ABB RAPID module: ProgSide1.mod

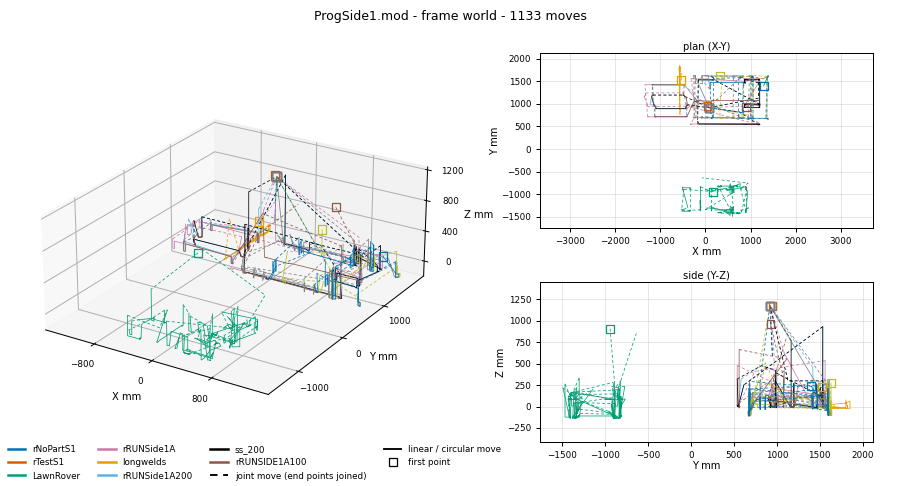
[picture p0: tool path of ProgSide1.mod in frame world, 1133 of 1133 moves have a stored position in this frame; points joined in program order, loops and branches not executed]
MODULE ProgSide1
	PERS bool bZ_B_onlySide2:=FALSE;
	PERS bool bZ_B_onlySide1:=FALSE;
	PERS bool bC_HalfstepSide2:=FALSE;
	PERS bool bC_HalfstepSide1:=FALSE;
	PERS bool bZ_HalfstepSide1:=FALSE;
	PERS bool bZ_HalfstepSide2:=FALSE;
	PERS bool bAngleSide1:=FALSE;
	PERS bool bAngleSide2:=FALSE;
	PERS bool bTestWeldSide1:=FALSE;
    PERS bool bTestWeldSide2:=FALSE;

    ! Boolian initialization for the SS 300 Frames
    PERS bool bNoPartSide1:=FALSE;
	PERS bool bNoPartSide2:=FALSE;
    PERS bool bPart1:=FALSE;
    PERS bool bPart2:=FALSE;
    PERS bool bPart3:=FALSE;
    PERS bool bPart4:=FALSE;
    PERS bool bPart5:=FALSE;
    PERS bool bPart6:=FALSE;
    PERS bool bPart7:=FALSE;
    PERS bool bPart8:=FALSE;
    PERS bool bPart9:=FALSE;
    PERS bool bPart10:=FALSE;
    PERS bool A_onlySide2:=FALSE;
    PERS bool B_onlySide2:=FALSE;
	PERS bool A_onlySide1:=TRUE;
    PERS bool B_onlySide1:=FALSE;
	PERS bool AB_Side1:=FALSE;
    PERS bool AB_Side2:=FALSE;

    ! Boolian initialization for the SelFrames procedures except the SS 300s.
    PERS bool bSkid50:=FALSE;
    PERS bool bSkid100:=FALSE;
	PERS bool bSkid200:=FALSE;
    PERS bool bSide1A100:=FALSE;
    PERS bool bSide1A200:=FALSE;

    PERS bool bRover:=TRUE;
    PERS bool bLongWeld:=FALSE;

    ! Boolian initialization for Parts menu selection.
    PERS bool bPart1:=FALSE;
    PERS bool bPart2:=FALSE;
    PERS bool bPart3:=FALSE;
    PERS bool bPart4:=FALSE;
    PERS bool bPart5:=FALSE;
    PERS bool bPart6:=FALSE;
    PERS bool bPart7:=FALSE;
    PERS bool bPart8:=FALSE;
    PERS bool bPart9:=FALSE;
    PERS bool bPart10:=FALSE;


	TASK PERS welddata weld7:=[15.24,16.6963,[7,0,0,0,0,0,0,0,0],[7,0,0,0,0,0,0,0,0]];
	TASK PERS welddata weld6:=[16.2983,16.6963,[6,0,0,0,0,0,0,0,0],[6,0,0,0,0,0,0,0,0]];

	CONST robtarget pPounceOS1:=[[-398.58,690.45,580.22],[0.00101632,0.999968,-0.00455572,0.00645523],[-1,0,-1,0],[9E+09,9E+09,9E+09,9E+09,9E+09,9E+09]];
	CONST robtarget pPounceS21:=[[580.19,77.23,83.43],[0.071601,0.767336,-0.436334,0.464416],[-1,0,-2,0],[9E+09,9E+09,9E+09,9E+09,9E+09,9E+09]];
	TASK PERS seamdata seam2:=[4,1,[1,0,52,74.0833,0,0,0,0,0],0,0,0,0,0,[1,0,48,0,0,0,0,0,0],0.01,0.1,[1,0,48,105.833,0,0,0,0,0],0,0,[0,0,0,0,0,0,0,0,0],1];
	TASK PERS seamdata seam10:=[4,1,[1,0,50,80.4333,0,0,0,0,0],0,0,0,0,0,[0,0,0,0,0,0,0,0,0],0.25,0.25,[1,0,50,38.1,0,0,0,0,0],0,0,[0,0,0,0,0,0,0,0,0],1];
	CONST robtarget pPounceS31:=[[358.52,159.10,437.93],[0.0181628,-0.398765,0.916866,0.00362624],[-2,0,-2,0],[9E+09,9E+09,9E+09,9E+09,9E+09,9E+09]];
	CONST robtarget pPounceS41:=[[193.25,136.11,113.74],[0.188325,0.84715,-0.195157,0.45693],[-1,-1,-2,0],[9E+09,9E+09,9E+09,9E+09,9E+09,9E+09]];
	PERS welddata weld11:=[13.5467,0,[1,0,50,84.6667,0,0,0,0,0],[0,0,0,0,0,0,0,0,0]];
	PERS welddata weld10:=[14.8167,0,[1,0,50,95.25,0,0,0,0,0],[0,0,0,0,0,0,0,0,0]];
	TASK PERS seamdata seam11:=[1,1,[1,0,50,84.6667,0,0,0,0,0],0,0,0,0,0,[0,0,0,0,0,0,0,0,0],0,0,[0,0,0,0,0,0,0,0,0],0,0,[0,0,0,0,0,0,0,0,0],0];
	TASK PERS seamdata seam12:=[1,1,[1,0,18.5,381,0,0,0,0,0],0,0,0,0,0,[0,0,0,0,0,0,0,0,0],0,0,[0,0,0,0,0,0,0,0,0],0,0,[0,0,0,0,0,0,0,0,0],0];
	TASK PERS seamdata seam13:=[1,1,[1,0,14,127,0,0,0,0,0],0,0,0,0,0,[0,0,0,0,0,0,0,0,0],0,0,[0,0,0,0,0,0,0,0,0],0,0,[0,0,0,0,0,0,0,0,0],0];
	PERS welddata weld12:=[13.97,0,[1,0,50,84.6667,0,0,0,0,0],[0,0,0,0,0,0,0,0,0]];
	PERS welddata weld13:=[6.90033,0,[1,0,20,105.833,0,0,0,0,0],[0,0,0,0,0,0,0,0,0]];
	CONST robtarget pSafeS11:=[[-996.19,963.00,488.78],[0.0459907,-0.688393,0.722625,0.0425673],[1,-1,1,0],[9E+09,9E+09,9E+09,9E+09,9E+09,9E+09]];
	CONST robtarget pSafeS21:=[[-996.19,963.00,488.76],[0.0459983,-0.688397,0.722622,0.0425559],[1,-1,1,0],[9E+09,9E+09,9E+09,9E+09,9E+09,9E+09]];
	CONST robtarget pSafeS31:=[[506.44,675.04,711.34],[0.0314656,-0.935633,0.203865,-0.286426],[0,0,-2,0],[9E+09,9E+09,9E+09,9E+09,9E+09,9E+09]];
	CONST robtarget pSafeS41:=[[488.47,1091.24,654.25],[0.0459806,-0.688392,0.722627,0.0425664],[0,0,-1,0],[9E+09,9E+09,9E+09,9E+09,9E+09,9E+09]];
	CONST robtarget pSafeS51:=[[528.23,1196.89,528.24],[0.224235,-0.753625,-0.525201,-0.325471],[0,-1,-3,0],[9E+09,9E+09,9E+09,9E+09,9E+09,9E+09]];
	CONST robtarget pSafeS61:=[[597.29,1295.03,43.37],[0.191334,-0.732058,-0.538062,-0.371444],[0,-1,-2,0],[9E+09,9E+09,9E+09,9E+09,9E+09,9E+09]];
	CONST robtarget pSafeS71:=[[542.66,1322.39,535.75],[0.223485,-0.764556,-0.487458,-0.357621],[0,-1,-2,0],[9E+09,9E+09,9E+09,9E+09,9E+09,9E+09]];
	CONST robtarget pSafeS81:=[[542.66,1322.38,535.76],[0.223484,-0.764558,-0.487457,-0.35762],[0,-1,-2,0],[9E+09,9E+09,9E+09,9E+09,9E+09,9E+09]];
	CONST robtarget pPounceS51:=[[15.28,993.81,754.75],[0.277209,0.263034,-0.848831,-0.365313],[0,0,0,0],[9E+09,9E+09,9E+09,9E+09,9E+09,9E+09]];
	CONST robtarget pPounceS61:=[[649.55,1131.56,389.19],[0.45355,-0.00505177,-0.879595,-0.143459],[0,0,0,0],[9E+09,9E+09,9E+09,9E+09,9E+09,9E+09]];
	TASK PERS seamdata seam3:=[1,1,[1,0,35,84.6667,0,0,0,0,0],0,0,0,0,0,[1,0,48,0,0,0,0,0,0],0.01,0.1,[1,0,48,105.833,0,0,0,0,0],0,0,[0,0,0,0,0,0,0,0,0],1];
	CONST robtarget pSafeS101:=[[572.94,23.46,738.68],[0.0502756,-0.467207,-0.815726,-0.337314],[0,0,0,0],[9E+09,9E+09,9E+09,9E+09,9E+09,9E+09]];
	CONST robtarget pSafeS111:=[[877.74,-1.14,1156.39],[0.00629855,0.0017594,0.999979,-0.000494623],[0,-1,0,0],[9E+09,9E+09,9E+09,9E+09,9E+09,9E+09]];
	CONST robtarget pSafeS121:=[[877.74,-1.14,1156.39],[0.00629925,0.00175887,0.999979,-0.000492925],[0,-1,0,0],[9E+09,9E+09,9E+09,9E+09,9E+09,9E+09]];
	CONST robtarget pSafeS131:=[[865.02,1139.54,-19.77],[0.144708,-0.274627,0.931028,0.191903],[0,-2,2,0],[9E+09,9E+09,9E+09,9E+09,9E+09,9E+09]];
	CONST robtarget pSafeS141:=[[849.60,1148.97,-24.06],[0.00628216,0.00187497,0.999979,-0.000396021],[0,-1,1,0],[9E+09,9E+09,9E+09,9E+09,9E+09,9E+09]];
	CONST robtarget pSafeS151:=[[1007.97,1505.52,122.27],[0.0460025,-0.688387,0.722632,0.0425454],[0,1,-2,0],[9E+09,9E+09,9E+09,9E+09,9E+09,9E+09]];
	CONST robtarget pHomePos20:=[[365.14,988.92,-33.91],[0.0351389,-0.509982,-0.859022,-0.0276858],[0,-1,1,0],[9E+09,9E+09,9E+09,9E+09,9E+09,9E+09]];
	CONST robtarget pHomePos30:=[[365.15,979.87,-33.91],[0.0351433,-0.509968,-0.85903,-0.0276827],[0,-1,1,0],[9E+09,9E+09,9E+09,9E+09,9E+09,9E+09]];
	CONST robtarget pHomePos40:=[[365.14,979.87,-15.16],[0.0351385,-0.509986,-0.859019,-0.0276867],[0,-1,1,0],[9E+09,9E+09,9E+09,9E+09,9E+09,9E+09]];
	CONST robtarget pHomePos50:=[[433.12,979.73,-15.17],[0.0351369,-0.509964,-0.859032,-0.0276871],[0,-1,1,0],[9E+09,9E+09,9E+09,9E+09,9E+09,9E+09]];
	CONST robtarget pHomePos60:=[[430.57,978.47,-32.25],[0.0351433,-0.50998,-0.859023,-0.0276796],[0,-1,1,0],[9E+09,9E+09,9E+09,9E+09,9E+09,9E+09]];
	CONST robtarget pHomePos70:=[[430.57,978.46,-32.26],[0.0351393,-0.509989,-0.859017,-0.027681],[0,-1,1,0],[9E+09,9E+09,9E+09,9E+09,9E+09,9E+09]];
	CONST robtarget pHomePos80:=[[430.59,974.37,-32.26],[0.0351321,-0.50997,-0.859029,-0.0276862],[0,-1,1,0],[9E+09,9E+09,9E+09,9E+09,9E+09,9E+09]];
	CONST robtarget pHomePos90:=[[430.57,974.36,-24.94],[0.0351397,-0.509992,-0.859016,-0.0276799],[0,-1,1,0],[9E+09,9E+09,9E+09,9E+09,9E+09,9E+09]];
	CONST robtarget pHomePos100:=[[445.83,974.38,-24.94],[0.0351383,-0.509986,-0.859019,-0.0276863],[0,-1,1,0],[9E+09,9E+09,9E+09,9E+09,9E+09,9E+09]];
	CONST robtarget pHomePos110:=[[446.40,974.36,-32.29],[0.0351532,-0.510006,-0.859007,-0.0276708],[0,-1,1,0],[9E+09,9E+09,9E+09,9E+09,9E+09,9E+09]];
	CONST robtarget pHomePos120:=[[446.42,974.37,-32.29],[0.0351424,-0.509994,-0.859014,-0.0276814],[0,-1,1,0],[9E+09,9E+09,9E+09,9E+09,9E+09,9E+09]];
	CONST robtarget pSafeS12:=[[1424.79,-683.57,-13.74],[0.019551,0.168491,0.985501,-0.00412114],[-1,1,-2,0],[9E+09,9E+09,9E+09,9E+09,9E+09,9E+09]];
	CONST robtarget pSafeS22:=[[1462.93,-789.47,-110.40],[0.0637154,0.393325,0.863983,0.307846],[-1,1,-2,0],[9E+09,9E+09,9E+09,9E+09,9E+09,9E+09]];
	CONST robtarget pSafeS32:=[[1462.93,-821.54,-110.39],[0.0637158,0.39332,0.863986,0.307843],[-1,1,-2,0],[9E+09,9E+09,9E+09,9E+09,9E+09,9E+09]];
	CONST robtarget pSafeS42:=[[1462.93,-821.54,-110.39],[0.0637186,0.393326,0.863982,0.307849],[-1,1,-2,0],[9E+09,9E+09,9E+09,9E+09,9E+09,9E+09]];
	CONST robtarget pSafeS52:=[[1462.55,-1477.98,-107.56],[0.0637139,0.393324,0.863983,0.30785],[-1,0,-1,0],[9E+09,9E+09,9E+09,9E+09,9E+09,9E+09]];
	CONST robtarget pSafeS62:=[[1462.54,-1515.56,-107.57],[0.0637098,0.393325,0.863984,0.307846],[-1,0,-1,0],[9E+09,9E+09,9E+09,9E+09,9E+09,9E+09]];
	CONST robtarget pSafeS72:=[[1462.54,-1515.57,-107.57],[0.0637139,0.39333,0.86398,0.307849],[-1,0,-1,0],[9E+09,9E+09,9E+09,9E+09,9E+09,9E+09]];
	CONST robtarget pSafeS82:=[[1462.55,-1515.57,-6.77],[0.063723,0.393334,0.863975,0.307857],[-1,0,-1,0],[9E+09,9E+09,9E+09,9E+09,9E+09,9E+09]];
	CONST robtarget pSafeS161:=[[44.14,948.66,1172.82],[0.0459836,-0.688397,0.722622,0.0425714],[0,-1,0,0],[9E+09,9E+09,9E+09,9E+09,9E+09,9E+09]];
	CONST robtarget pSafeS171:=[[877.68,-1.12,1156.34],[0.00623811,0.00177345,0.999979,-0.000467886],[0,-1,0,0],[9E+09,9E+09,9E+09,9E+09,9E+09,9E+09]];
	CONST robtarget pSafeS181:=[[1178.99,1129.25,299.25],[0.0635535,0.517233,-0.779104,0.348467],[0,1,-3,1],[9E+09,9E+09,9E+09,9E+09,9E+09,9E+09]];
	CONST robtarget pSafeS191:=[[877.68,-1.12,1156.34],[0.00623811,0.00177268,0.999979,-0.000467882],[0,-1,0,0],[9E+09,9E+09,9E+09,9E+09,9E+09,9E+09]];
	CONST robtarget pSafeS201:=[[631.06,-50.80,790.98],[0.377429,-0.0153459,-0.925903,0.00402947],[-1,-1,-5,0],[9E+09,9E+09,9E+09,9E+09,9E+09,9E+09]];
	CONST robtarget pSafeS211:=[[631.06,-50.80,790.98],[0.377429,-0.0153486,-0.925903,0.00403031],[-1,-1,-5,0],[9E+09,9E+09,9E+09,9E+09,9E+09,9E+09]];


!XXXXXXXXXXXXXXXXXXXXXXXXXXXXXXXXXXXXXXXXXXXXXXXXXXXXXXXXXXXX

!XXXXXXXXXXXXXXXXXXXXXXXXXXXXXXXXXXXXXXXXXXXXXXXXXXXXXXXXXXXX
!xxxxxxxxxxxxxxxxxxxxxxxxxxxxxxxxxxxxxxxxxxxxxxxxxxxxxxxxxxxxxxxx




	PROC rNoPartS1()
		MoveJ pSafeS1, v800, fine, tWeldGun;
		MoveJ pPounceS1, v800, fine, tWeldGun;
		MoveJ pSafeS1, v800, fine, tWeldGun;
	ENDPROC
	PROC rTstA1()
		TPWrite "A S1";
	ENDPROC
	PROC rTstB1()
		TPWrite "B S1";
	ENDPROC
	PROC rTestS1()
		MoveJ [[44.14,948.66,1172.81],[0.0459874,-0.688394,0.722625,0.042569],[0,-1,0,0],[9E+09,9E+09,9E+09,9E+09,9E+09,9E+09]], v1000, z50, tWeldGun;
	ENDPROC
	PROC LawnRover()
		rTestPosTop;
		TPWrite "Side 1 B";
		MoveJ [[173.01,-945.09,908.66],[0.230148,-0.640466,-0.674994,-0.284991],[-1,0,0,0],[9E+09,9E+09,9E+09,9E+09,9E+09,9E+09]], vmax, z50, tWeldGun;
		MoveJ [[-516.56,-891.88,262.76],[0.200577,-0.67934,-0.672798,-0.213563],[-2,0,-1,0],[9E+09,9E+09,9E+09,9E+09,9E+09,9E+09]], vmax, z10, tWeldGun;
		MoveL [[-514.49,-897.92,-127.68],[0.230166,-0.665843,-0.672051,-0.22809],[-2,0,-1,0],[9E+09,9E+09,9E+09,9E+09,9E+09,9E+09]], vmax, z10, tWeldGun;
		ArcLStart [[-513.42,-896.95,-136.62],[0.210767,-0.657306,-0.686363,-0.228983],[-2,0,-1,0],[9E+09,9E+09,9E+09,9E+09,9E+09,9E+09]], v50, seam13, weld13\Weave:=weave1, fine, tWeldGun;
		ArcLEnd [[-481.07,-897.11,-138.20],[0.210746,-0.657346,-0.686325,-0.229001],[-2,0,-1,0],[9E+09,9E+09,9E+09,9E+09,9E+09,9E+09]], v5, seam13, weld13\Weave:=weave1, fine, tWeldGun;
		MoveL [[-479.64,-891.87,-91.90],[0.200495,-0.679391,-0.672743,-0.213649],[-2,0,-1,0],[9E+09,9E+09,9E+09,9E+09,9E+09,9E+09]], vmax, z10, tWeldGun;
		MoveJ [[-526.59,-1340.74,-77.97],[0.272049,0.539222,-0.749573,0.270868],[-2,0,-3,0],[9E+09,9E+09,9E+09,9E+09,9E+09,9E+09]], vmax, z10, tWeldGun;
		MoveL [[-519.95,-1336.21,-124.59],[0.179682,0.6848,-0.680507,0.188877],[-2,-1,-3,0],[9E+09,9E+09,9E+09,9E+09,9E+09,9E+09]], vmax, z10, tWeldGun;
		ArcLStart [[-521.69,-1337.70,-132.47],[0.193399,0.681112,-0.684086,0.175244],[-2,-1,-3,0],[9E+09,9E+09,9E+09,9E+09,9E+09,9E+09]], v50, seam13, weld13\Weave:=weave1, fine, tWeldGun;
		ArcLEnd [[-490.93,-1337.53,-132.49],[0.193282,0.681205,-0.684029,0.175234],[-2,-1,-3,0],[9E+09,9E+09,9E+09,9E+09,9E+09,9E+09]], v5, seam13, weld13\Weave:=weave1, fine, tWeldGun;
		MoveL [[-484.84,-1342.71,46.50],[0.235633,0.655478,-0.679432,0.230648],[-2,-1,-3,0],[9E+09,9E+09,9E+09,9E+09,9E+09,9E+09]], vmax, z10, tWeldGun;
		MoveJ [[-392.56,-1296.67,69.52],[0.264192,0.731229,-0.303703,0.550702],[-2,0,0,0],[9E+09,9E+09,9E+09,9E+09,9E+09,9E+09]], vmax, z20, tWeldGun;
		MoveL [[-512.18,-856.47,-124.70],[0.238884,-0.653044,-0.673688,-0.250226],[-2,0,-1,0],[9E+09,9E+09,9E+09,9E+09,9E+09,9E+09]], vmax, z10, tWeldGun;
		ArcLStart [[-513.54,-858.91,-136.72],[0.215398,-0.662814,-0.680722,-0.225612],[-2,0,-1,0],[9E+09,9E+09,9E+09,9E+09,9E+09,9E+09]], v50, seam13, weld13, fine, tWeldGun;
		!ArcLEnd [[-473.42,-859.48,-137.35],[0.215439,-0.662758,-0.68077,-0.22559],[-2,0,-1,0],[9E+09,9E+09,9E+09,9E+09,9E+09,9E+09]], v5, seam13, weld13\Weave:=weave1, fine, tWeldGun;
		!MoveL [[-470.56,-868.46,-128.98],[0.215449,-0.66272,-0.680808,-0.225579],[-2,0,-1,0],[9E+09,9E+09,9E+09,9E+09,9E+09,9E+09]], vmax, z10, tWeldGun;
		!MoveL [[-436.87,-865.82,-129.01],[0.215414,-0.662677,-0.680771,-0.225849],[-2,0,-1,0],[9E+09,9E+09,9E+09,9E+09,9E+09,9E+09]], vmax, z10, tWeldGun;
		!ArcLStart [[-436.92,-859.84,-136.80],[0.215444,-0.662646,-0.680803,-0.225813],[-2,0,-1,0],[9E+09,9E+09,9E+09,9E+09,9E+09,9E+09]], v50, seam13, weld13\Weave:=weave1, fine, tWeldGun;
		!ArcLEnd [[-395.30,-860.19,-135.58],[0.21546,-0.662716,-0.680804,-0.225593],[-2,0,-1,0],[9E+09,9E+09,9E+09,9E+09,9E+09,9E+09]], v5, seam13, weld13\Weave:=weave1, fine, tWeldGun;
		!MoveL [[-394.28,-872.79,-127.38],[0.215463,-0.66272,-0.6808,-0.225589],[-2,0,-1,0],[9E+09,9E+09,9E+09,9E+09,9E+09,9E+09]], vmax, z10, tWeldGun;
		!MoveL [[-366.90,-866.62,-125.77],[0.215457,-0.662713,-0.680808,-0.225591],[-2,0,-1,0],[9E+09,9E+09,9E+09,9E+09,9E+09,9E+09]], vmax, z10, tWeldGun;
		!ArcLStart [[-366.93,-860.65,-137.16],[0.215461,-0.662729,-0.680792,-0.225588],[-2,0,-1,0],[9E+09,9E+09,9E+09,9E+09,9E+09,9E+09]], v50, seam13, weld13\Weave:=weave1, fine, tWeldGun;
		ArcLEnd [[-338.32,-860.21,-136.79],[0.215451,-0.662739,-0.68078,-0.225604],[-2,0,-1,0],[9E+09,9E+09,9E+09,9E+09,9E+09,9E+09]], v5, seam13, weld13\Weave:=weave1, fine, tWeldGun;
		MoveL [[-339.56,-873.86,-125.98],[0.215452,-0.662777,-0.680806,-0.225413],[-2,0,-1,0],[9E+09,9E+09,9E+09,9E+09,9E+09,9E+09]], vmax, z10, tWeldGun;
		MoveL [[-336.25,-871.19,-128.23],[0.0916487,-0.841258,-0.420907,-0.326687],[-2,0,-1,0],[9E+09,9E+09,9E+09,9E+09,9E+09,9E+09]], vmax, z10, tWeldGun;
		ArcLStart [[-338.59,-862.58,-134.25],[0.091653,-0.841261,-0.420909,-0.326675],[-2,0,-1,0],[9E+09,9E+09,9E+09,9E+09,9E+09,9E+09]], v50, seam13, weld13, fine, tWeldGun;
		ArcLEnd [[-343.89,-887.38,-134.91],[0.00905831,0.920106,0.0370212,0.389812],[-2,0,0,0],[9E+09,9E+09,9E+09,9E+09,9E+09,9E+09]], v5, seam13, weld13, fine, tWeldGun;
		MoveL [[-340.52,-888.78,-94.76],[0.0606807,0.91536,0.0671192,0.392339],[-2,0,0,0],[9E+09,9E+09,9E+09,9E+09,9E+09,9E+09]], v100, z10, tWeldGun;
		!MoveL [[-322.29,-862.50,-115.71],[0.124255,-0.837706,-0.434858,-0.306118],[-2,0,0,0],[9E+09,9E+09,9E+09,9E+09,9E+09,9E+09]], v100, z10, tWeldGun;
		!ArcLStart [[-317.89,-862.07,-130.90],[0.120916,-0.838204,-0.433585,-0.307894],[-2,0,0,0],[9E+09,9E+09,9E+09,9E+09,9E+09,9E+09]], v40, seam13, weld13\Weave:=weave1, fine, tWeldGun;
		!ArcLEnd [[-340.01,-859.38,-134.88],[0.124327,-0.837704,-0.434755,-0.306241],[-2,0,0,0],[9E+09,9E+09,9E+09,9E+09,9E+09,9E+09]], v5, seam13, weld13\Weave:=weave1, fine, tWeldGun;
		MoveL [[-337.89,-880.77,33.09],[0.124309,-0.837706,-0.434822,-0.306146],[-2,0,0,0],[9E+09,9E+09,9E+09,9E+09,9E+09,9E+09]], vmax, z10, tWeldGun;
		MoveJ [[-332.34,-1363.85,48.88],[0.219066,0.836756,-0.390875,0.31475],[-2,-1,1,0],[9E+09,9E+09,9E+09,9E+09,9E+09,9E+09]], vmax, z10, tWeldGun;
		MoveL [[-348.32,-1358.04,-125.11],[0.0288552,0.954843,-0.0190534,0.295092],[-2,-1,1,0],[9E+09,9E+09,9E+09,9E+09,9E+09,9E+09]], vmax, z10, tWeldGun;
		ArcLStart [[-348.85,-1357.02,-134.12],[0.0288204,0.95485,-0.0190118,0.295075],[-2,-1,1,0],[9E+09,9E+09,9E+09,9E+09,9E+09,9E+09]], v50, seam13, weld13\Weave:=weave1, fine, tWeldGun;
		ArcLEnd [[-348.77,-1383.12,-133.63],[0.144948,0.917185,-0.235244,0.287092],[-2,-1,1,0],[9E+09,9E+09,9E+09,9E+09,9E+09,9E+09]], v5, seam13, weld13\Weave:=weave1, fine, tWeldGun;
		MoveL [[-352.02,-1382.79,-125.00],[0.145009,0.917103,-0.235465,0.287142],[-2,-1,1,0],[9E+09,9E+09,9E+09,9E+09,9E+09,9E+09]], vmax, z10, tWeldGun;
		!MoveL [[-328.65,-1384.41,-121.55],[0.145003,0.917127,-0.235391,0.287129],[-2,-1,1,0],[9E+09,9E+09,9E+09,9E+09,9E+09,9E+09]], vmax, z10, tWeldGun;
		!ArcLStart [[-329.96,-1384.26,-128.86],[0.144876,0.917192,-0.23532,0.287045],[-2,-1,1,0],[9E+09,9E+09,9E+09,9E+09,9E+09,9E+09]], v40, seam13, weld13\Weave:=weave1, fine, tWeldGun;
		!ArcLEnd [[-349.04,-1384.95,-130.97],[0.144974,0.917151,-0.235337,0.287113],[-2,-1,1,0],[9E+09,9E+09,9E+09,9E+09,9E+09,9E+09]], v5, seam13, weld13\Weave:=weave1, fine, tWeldGun;
		!MoveL [[-350.83,-1367.95,-122.57],[0.144998,0.917131,-0.235387,0.287125],[-2,-1,1,0],[9E+09,9E+09,9E+09,9E+09,9E+09,9E+09]], vmax, z10, tWeldGun;
		MoveL [[-341.99,-1371.18,-117.57],[0.232266,0.668561,-0.669899,0.224308],[-2,-1,1,0],[9E+09,9E+09,9E+09,9E+09,9E+09,9E+09]], vmax, z10, tWeldGun;
		ArcLStart [[-346.14,-1380.75,-134.00],[0.232258,0.668629,-0.669841,0.22429],[-2,-1,1,0],[9E+09,9E+09,9E+09,9E+09,9E+09,9E+09]], v30, seam13, weld13, fine, tWeldGun;
		!ArcLEnd [[-381.42,-1380.96,-134.98],[0.232253,0.668599,-0.669868,0.2243],[-2,-1,1,0],[9E+09,9E+09,9E+09,9E+09,9E+09,9E+09]], v5, seam13, weld13, fine, tWeldGun;
		!MoveL [[-381.43,-1374.36,-128.77],[0.232262,0.668602,-0.669863,0.224299],[-2,-1,1,0],[9E+09,9E+09,9E+09,9E+09,9E+09,9E+09]], vmax, z10, tWeldGun;
		!MoveL [[-417.42,-1374.56,-128.76],[0.232259,0.668611,-0.669855,0.224298],[-2,-1,1,0],[9E+09,9E+09,9E+09,9E+09,9E+09,9E+09]], vmax, z10, tWeldGun;
		!ArcLStart [[-417.85,-1379.53,-134.58],[0.215828,0.673878,-0.675969,0.205846],[-2,-1,1,0],[9E+09,9E+09,9E+09,9E+09,9E+09,9E+09]], v50, seam13, weld13\Weave:=weave1, fine, tWeldGun;
		!ArcLEnd [[-443.05,-1379.79,-134.59],[0.215834,0.673901,-0.675942,0.205854],[-2,-1,1,0],[9E+09,9E+09,9E+09,9E+09,9E+09,9E+09]], v5, seam13, weld13\Weave:=weave1, fine, tWeldGun;
		!MoveL [[-444.47,-1371.57,-127.54],[0.232274,0.66863,-0.669834,0.224288],[-2,-1,1,0],[9E+09,9E+09,9E+09,9E+09,9E+09,9E+09]], vmax, z10, tWeldGun;
		!MoveL [[-474.23,-1371.36,-127.53],[0.232273,0.668635,-0.66983,0.224288],[-2,-1,1,0],[9E+09,9E+09,9E+09,9E+09,9E+09,9E+09]], vmax, z10, tWeldGun;
		!ArcLStart [[-474.48,-1379.73,-135.16],[0.232264,0.668658,-0.669815,0.224273],[-2,-1,1,0],[9E+09,9E+09,9E+09,9E+09,9E+09,9E+09]], v50, seam13, weld13\Weave:=weave1, fine, tWeldGun;
		ArcLEnd [[-520.49,-1380.63,-135.80],[0.232194,0.668749,-0.669754,0.224259],[-2,-1,1,0],[9E+09,9E+09,9E+09,9E+09,9E+09,9E+09]], v5, seam13, weld13\Weave:=weave1, fine, tWeldGun;
		MoveL [[-521.34,-1368.99,120.05],[0.232497,0.668664,-0.669682,0.22441],[-2,-1,1,0],[9E+09,9E+09,9E+09,9E+09,9E+09,9E+09]], vmax, z10, tWeldGun;
		MoveJ [[-94.49,-1349.72,64.27],[0.311518,0.0288903,-0.949685,-0.0148846],[-2,0,-2,0],[9E+09,9E+09,9E+09,9E+09,9E+09,9E+09]], vmax, z10, tWeldGun;
		MoveJ [[-121.47,-1146.91,200.07],[0.233067,0.684788,-0.672515,-0.156426],[-1,-1,-2,0],[9E+09,9E+09,9E+09,9E+09,9E+09,9E+09]], vmax, z10, tWeldGun;
		MoveL [[-117.16,-1374.82,-109.86],[0.220566,0.688799,-0.675571,-0.143216],[-1,-1,-2,0],[9E+09,9E+09,9E+09,9E+09,9E+09,9E+09]], vmax, z10, tWeldGun;
		ArcLStart [[-117.21,-1374.86,-121.15],[0.220636,0.688785,-0.675564,-0.143209],[-1,-1,-2,0],[9E+09,9E+09,9E+09,9E+09,9E+09,9E+09]], v50, seam13, weld13\Weave:=weave1, fine, tWeldGun;
		ArcLEnd [[-117.25,-1343.15,-121.11],[0.220558,0.688816,-0.67554,-0.143296],[-1,-1,-2,0],[9E+09,9E+09,9E+09,9E+09,9E+09,9E+09]], v5, seam13, weld13\Weave:=weave1, fine, tWeldGun;
		MoveL [[-112.47,-1343.13,-110.12],[0.220583,0.6888,-0.675545,-0.143308],[-1,-1,-2,0],[9E+09,9E+09,9E+09,9E+09,9E+09,9E+09]], vmax, z10, tWeldGun;
		MoveL [[-112.47,-861.36,-110.12],[0.220582,0.688805,-0.67554,-0.143307],[-1,-1,-2,0],[9E+09,9E+09,9E+09,9E+09,9E+09,9E+09]], vmax, z10, tWeldGun;
		ArcLStart [[-114.29,-865.15,-124.72],[0.220598,0.688808,-0.675528,-0.143326],[-1,-1,-2,0],[9E+09,9E+09,9E+09,9E+09,9E+09,9E+09]], v50, seam13, weld13\Weave:=weave1, fine, tWeldGun;
		ArcLEnd [[-114.32,-834.89,-124.92],[0.220557,0.688836,-0.675507,-0.143359],[-1,-1,-2,0],[9E+09,9E+09,9E+09,9E+09,9E+09,9E+09]], v5, seam13, weld13\Weave:=weave1, fine, tWeldGun;
		MoveL [[-108.44,-837.80,142.79],[0.0521127,0.721407,-0.690258,0.0200149],[-2,-1,-3,0],[9E+09,9E+09,9E+09,9E+09,9E+09,9E+09]], vmax, z10, tWeldGun;
		MoveJ [[5.08,-892.16,87.65],[0.246917,-0.649526,-0.670091,-0.261011],[-2,0,-1,0],[9E+09,9E+09,9E+09,9E+09,9E+09,9E+09]], vmax, z10, tWeldGun;
		MoveL [[5.70,-898.13,-125.58],[0.246931,-0.64953,-0.670081,-0.261012],[-2,0,-1,0],[9E+09,9E+09,9E+09,9E+09,9E+09,9E+09]], vmax, z10, tWeldGun;
		ArcLStart [[5.30,-897.90,-137.78],[0.203047,-0.669211,-0.681329,-0.216148],[-2,0,-1,0],[9E+09,9E+09,9E+09,9E+09,9E+09,9E+09]], v50, seam13, weld13\Weave:=weave1, fine, tWeldGun;
		ArcLEnd [[39.29,-898.07,-137.00],[0.203054,-0.669216,-0.681319,-0.216158],[-1,0,-1,0],[9E+09,9E+09,9E+09,9E+09,9E+09,9E+09]], v5, seam13, weld13\Weave:=weave1, fine, tWeldGun;
		MoveL [[40.66,-920.62,70.48],[0.246699,-0.649617,-0.670207,-0.260692],[-1,0,-1,0],[9E+09,9E+09,9E+09,9E+09,9E+09,9E+09]], vmax, z10, tWeldGun;
		MoveJ [[283.83,-931.65,13.13],[0.246958,-0.649486,-0.670134,-0.26096],[-1,0,0,0],[9E+09,9E+09,9E+09,9E+09,9E+09,9E+09]], vmax, z10, tWeldGun;
		MoveL [[286.40,-910.85,-115.99],[0.24696,-0.649475,-0.670149,-0.260949],[-1,0,0,0],[9E+09,9E+09,9E+09,9E+09,9E+09,9E+09]], vmax, z10, tWeldGun;
		ArcLStart [[287.09,-901.24,-138.12],[0.20011,-0.665429,-0.68641,-0.214478],[-1,-1,0,0],[9E+09,9E+09,9E+09,9E+09,9E+09,9E+09]], v50, seam13, weld13\Weave:=weave1, fine, tWeldGun;
		ArcLEnd [[319.26,-901.70,-138.51],[0.200189,-0.665343,-0.686488,-0.214425],[-1,-1,0,0],[9E+09,9E+09,9E+09,9E+09,9E+09,9E+09]], v5, seam13, weld13\Weave:=weave1, fine, tWeldGun;
		MoveL [[324.35,-903.06,-116.80],[0.246972,-0.649396,-0.670267,-0.260831],[-1,0,0,0],[9E+09,9E+09,9E+09,9E+09,9E+09,9E+09]], vmax, z10, tWeldGun;
		MoveJ [[559.57,-898.83,-116.82],[0.246966,-0.649476,-0.670148,-0.260944],[-1,-1,0,0],[9E+09,9E+09,9E+09,9E+09,9E+09,9E+09]], vmax, z10, tWeldGun;
		MoveL [[566.73,-906.53,-132.43],[0.246936,-0.649457,-0.670181,-0.260932],[-1,-1,0,0],[9E+09,9E+09,9E+09,9E+09,9E+09,9E+09]], vmax, z10, tWeldGun;
		ArcLStart [[564.18,-902.64,-136.45],[0.203779,-0.664669,-0.684636,-0.219006],[-1,-1,0,0],[9E+09,9E+09,9E+09,9E+09,9E+09,9E+09]], v50, seam13, weld13\Weave:=weave1, fine, tWeldGun;
		ArcLEnd [[595.80,-903.83,-135.82],[0.203773,-0.664709,-0.684589,-0.219037],[-1,-1,0,0],[9E+09,9E+09,9E+09,9E+09,9E+09,9E+09]], v5, seam13, weld13\Weave:=weave1, fine, tWeldGun;
		MoveL [[596.75,-960.43,-56.34],[0.246991,-0.649449,-0.670174,-0.260919],[-1,-1,0,0],[9E+09,9E+09,9E+09,9E+09,9E+09,9E+09]], vmax, z10, tWeldGun;
		MoveJ [[601.82,-903.83,-123.32],[0.326164,-0.613251,-0.630337,-0.346722],[-1,0,0,0],[9E+09,9E+09,9E+09,9E+09,9E+09,9E+09]], vmax, z10, tWeldGun;
		MoveL [[598.73,-903.81,-136.04],[0.274721,-0.639021,-0.654339,-0.296685],[-1,0,0,0],[9E+09,9E+09,9E+09,9E+09,9E+09,9E+09]], v100, z10, tWeldGun;
		ArcLStart [[599.82,-898.69,-137.04],[0.274731,-0.639021,-0.654342,-0.296669],[-1,0,0,0],[9E+09,9E+09,9E+09,9E+09,9E+09,9E+09]], v40, seam13, weld13\Weave:=weave1, fine, tWeldGun;
		ArcLEnd [[632.81,-898.75,-137.05],[0.274699,-0.639022,-0.654363,-0.296649],[-1,0,0,0],[9E+09,9E+09,9E+09,9E+09,9E+09,9E+09]], v5, seam13, weld13\Weave:=weave1, fine, tWeldGun;
		MoveL [[633.74,-910.04,-132.93],[0.326202,-0.613258,-0.630325,-0.346695],[-1,0,0,0],[9E+09,9E+09,9E+09,9E+09,9E+09,9E+09]], vmax, z10, tWeldGun;
		MoveL [[633.73,-910.04,183.03],[0.326216,-0.613247,-0.630334,-0.346685],[-1,0,0,0],[9E+09,9E+09,9E+09,9E+09,9E+09,9E+09]], vmax, z10, tWeldGun;
		MoveJ [[627.00,-822.44,298.30],[0.361159,0.600904,-0.609737,0.36973],[-1,-1,-2,0],[9E+09,9E+09,9E+09,9E+09,9E+09,9E+09]], vmax, z10, tWeldGun;
		MoveL [[627.73,-843.08,-138.79],[0.402411,0.574308,-0.586575,0.405173],[-1,-2,-1,0],[9E+09,9E+09,9E+09,9E+09,9E+09,9E+09]], vmax, z10, tWeldGun;
		ArcLStart [[625.49,-849.82,-138.90],[0.402522,0.574183,-0.586614,0.405185],[-1,-2,-1,0],[9E+09,9E+09,9E+09,9E+09,9E+09,9E+09]], v50, seam13, weld13\Weave:=weave1, fine, tWeldGun;
		ArcLEnd [[591.69,-849.46,-138.90],[0.402522,0.574182,-0.586613,0.405187],[-1,-2,-1,0],[9E+09,9E+09,9E+09,9E+09,9E+09,9E+09]], v5, seam13, weld13\Weave:=weave1, fine, tWeldGun;
		MoveL [[595.98,-827.09,-135.34],[0.402393,0.574513,-0.586267,0.405347],[-1,-2,-1,0],[9E+09,9E+09,9E+09,9E+09,9E+09,9E+09]], vmax, z10, tWeldGun;
		MoveL [[627.09,-846.85,78.98],[0.483059,0.507565,-0.528798,0.478963],[-1,-2,-1,0],[9E+09,9E+09,9E+09,9E+09,9E+09,9E+09]], vmax, z10, tWeldGun;
		ArcLStart [[623.92,-856.82,80.37],[0.483064,0.507539,-0.52884,0.478939],[-1,-2,-1,0],[9E+09,9E+09,9E+09,9E+09,9E+09,9E+09]], v40, seam13, weld13\Weave:=weave1, fine, tWeldGun;
		ArcLEnd [[590.91,-852.32,80.98],[0.483106,0.507553,-0.528792,0.478934],[-1,-2,-1,0],[9E+09,9E+09,9E+09,9E+09,9E+09,9E+09]], v5, seam13, weld13\Weave:=weave1, fine, tWeldGun;
		MoveL [[594.84,-840.41,79.51],[0.487671,0.503288,-0.532967,0.474157],[-1,-2,-1,0],[9E+09,9E+09,9E+09,9E+09,9E+09,9E+09]], vmax, z10, tWeldGun;
		SingArea\Wrist;
		MoveJ [[510.38,-859.01,160.69],[0.00485322,0.746032,-0.024255,0.665452],[-1,0,0,0],[9E+09,9E+09,9E+09,9E+09,9E+09,9E+09]], vmax, z10, tWeldGun;
		MoveL [[590.96,-857.11,78.44],[0.00482135,0.745929,-0.024224,0.665567],[-1,0,0,0],[9E+09,9E+09,9E+09,9E+09,9E+09,9E+09]], vmax, z10, tWeldGun;
		ArcLStart [[595.46,-855.56,78.39],[0.00479068,0.745947,-0.0242061,0.665549],[-1,0,0,0],[9E+09,9E+09,9E+09,9E+09,9E+09,9E+09]], v40, seam13, weld13\Weave:=weave1, fine, tWeldGun;
		ArcLEnd [[594.74,-887.31,78.36],[0.00476122,0.74597,-0.0241871,0.665524],[-1,0,0,0],[9E+09,9E+09,9E+09,9E+09,9E+09,9E+09]], v5, seam13, weld13\Weave:=weave1, fine, tWeldGun;
		MoveL [[545.64,-889.59,83.73],[0.0047987,0.745982,-0.0242261,0.665508],[-1,0,0,0],[9E+09,9E+09,9E+09,9E+09,9E+09,9E+09]], vmax, z10, tWeldGun;
		MoveL [[545.47,-1007.73,83.69],[0.00477345,0.745999,-0.0242032,0.665491],[-1,0,0,0],[9E+09,9E+09,9E+09,9E+09,9E+09,9E+09]], vmax, z10, tWeldGun;
		MoveJ [[631.13,-962.99,83.64],[0.467638,-0.538268,-0.512971,-0.477958],[-1,0,0,0],[9E+09,9E+09,9E+09,9E+09,9E+09,9E+09]], vmax, z10, tWeldGun;
		MoveL [[598.78,-893.01,80.08],[0.467241,-0.531733,-0.519718,-0.478373],[-1,0,0,0],[9E+09,9E+09,9E+09,9E+09,9E+09,9E+09]], vmax, z10, tWeldGun;
		ArcLStart [[597.51,-884.44,80.09],[0.467289,-0.531729,-0.519697,-0.478352],[-1,0,0,0],[9E+09,9E+09,9E+09,9E+09,9E+09,9E+09]], v50, seam13, weld13\Weave:=weave1, fine, tWeldGun;
		ArcLEnd [[628.34,-885.62,79.45],[0.467277,-0.53174,-0.519666,-0.478386],[-1,0,0,0],[9E+09,9E+09,9E+09,9E+09,9E+09,9E+09]], v5, seam13, weld13\Weave:=weave1, fine, tWeldGun;
		MoveL [[633.84,-953.29,84.81],[0.467086,-0.531839,-0.51974,-0.478381],[-1,0,0,0],[9E+09,9E+09,9E+09,9E+09,9E+09,9E+09]], vmax, z10, tWeldGun;
		MoveJ [[-0.34,-1346.80,171.20],[0.287604,0.644423,-0.651566,0.278325],[-1,-1,-2,0],[9E+09,9E+09,9E+09,9E+09,9E+09,9E+09]], vmax, z10, tWeldGun;
		MoveL [[-2.14,-1338.76,-121.61],[0.287464,0.644565,-0.651541,0.278198],[-1,-1,-2,0],[9E+09,9E+09,9E+09,9E+09,9E+09,9E+09]], vmax, z10, tWeldGun;
		ArcLStart [[-0.59,-1345.37,-136.31],[0.245261,0.661538,-0.666169,0.241731],[-1,0,-2,0],[9E+09,9E+09,9E+09,9E+09,9E+09,9E+09]], v40, seam13, weld13\Weave:=weave1, fine, tWeldGun;
		ArcLEnd [[34.33,-1344.96,-135.32],[0.245262,0.661569,-0.666134,0.241742],[-1,0,-2,0],[9E+09,9E+09,9E+09,9E+09,9E+09,9E+09]], v5, seam13, weld13\Weave:=weave1, fine, tWeldGun;
		MoveL [[33.45,-1306.76,35.10],[0.287609,0.644475,-0.651512,0.278328],[-1,-1,-2,0],[9E+09,9E+09,9E+09,9E+09,9E+09,9E+09]], vmax, z10, tWeldGun;
		MoveL [[273.41,-1327.02,35.12],[0.287608,0.6445,-0.651487,0.278327],[-1,-1,-2,0],[9E+09,9E+09,9E+09,9E+09,9E+09,9E+09]], vmax, z10, tWeldGun;
		MoveL [[281.49,-1342.97,-129.04],[0.226085,0.668734,-0.671173,0.226292],[-1,0,-2,0],[9E+09,9E+09,9E+09,9E+09,9E+09,9E+09]], vmax, z10, tWeldGun;
		ArcLStart [[279.86,-1346.54,-134.30],[0.226103,0.668741,-0.671174,0.226249],[-1,0,-2,0],[9E+09,9E+09,9E+09,9E+09,9E+09,9E+09]], v40, seam13, weld13\Weave:=weave1, fine, tWeldGun;
		ArcLEnd [[313.73,-1346.47,-133.85],[0.216577,0.67052,-0.675561,0.217062],[-1,0,-2,0],[9E+09,9E+09,9E+09,9E+09,9E+09,9E+09]], v5, seam13, weld13\Weave:=weave1, fine, tWeldGun;
		MoveL [[313.56,-1350.36,-117.72],[0.287596,0.644518,-0.651477,0.278324],[-1,-1,-2,0],[9E+09,9E+09,9E+09,9E+09,9E+09,9E+09]], vmax, z10, tWeldGun;
		MoveL [[559.03,-1342.37,-128.81],[0.261338,0.655204,-0.662463,0.2521],[-1,0,-2,0],[9E+09,9E+09,9E+09,9E+09,9E+09,9E+09]], vmax, z10, tWeldGun;
		ArcLStart [[559.48,-1347.56,-134.32],[0.242704,0.66214,-0.669449,0.233462],[-1,0,-2,0],[9E+09,9E+09,9E+09,9E+09,9E+09,9E+09]], v40, seam13, weld13\Weave:=weave1, fine, tWeldGun;
		ArcLEnd [[590.72,-1348.56,-134.75],[0.242689,0.662054,-0.669527,0.233498],[-1,0,-2,0],[9E+09,9E+09,9E+09,9E+09,9E+09,9E+09]], v5, seam13, weld13\Weave:=weave1, fine, tWeldGun;
		MoveL [[591.10,-1294.92,-96.48],[0.287644,0.644544,-0.6514,0.278391],[-1,-1,-2,0],[9E+09,9E+09,9E+09,9E+09,9E+09,9E+09]], vmax, z10, tWeldGun;
		MoveL [[591.39,-1347.13,-134.61],[0.309685,0.644241,-0.632283,0.298777],[-1,-1,-2,0],[9E+09,9E+09,9E+09,9E+09,9E+09,9E+09]], vmax, z10, tWeldGun;
		ArcLStart [[596.97,-1352.85,-136.25],[0.320366,0.639208,-0.626493,0.310301],[-1,-1,-2,0],[9E+09,9E+09,9E+09,9E+09,9E+09,9E+09]], v40, seam13, weld13\Weave:=weave1, fine, tWeldGun;
		ArcLEnd [[621.87,-1354.95,-137.78],[0.327716,0.635456,-0.623102,0.317085],[-1,-1,-2,0],[9E+09,9E+09,9E+09,9E+09,9E+09,9E+09]], v5, seam13, weld13\Weave:=weave1, fine, tWeldGun;
		MoveL [[594.26,-1304.04,-124.90],[0.375061,0.603881,-0.605571,0.35769],[-1,-1,-2,0],[9E+09,9E+09,9E+09,9E+09,9E+09,9E+09]], vmax, z10, tWeldGun;
		MoveL [[623.93,-1279.28,49.33],[0.327728,0.635484,-0.623033,0.31715],[-1,-1,-2,0],[9E+09,9E+09,9E+09,9E+09,9E+09,9E+09]], vmax, z10, tWeldGun;
		MoveJ [[598.90,-1494.47,216.89],[0.17643,-0.701594,-0.668329,-0.173135],[-1,-1,0,0],[9E+09,9E+09,9E+09,9E+09,9E+09,9E+09]], vmax, z10, tWeldGun;
		MoveL [[597.59,-1416.16,-134.75],[0.380292,-0.610593,-0.58263,-0.378282],[-1,0,0,0],[9E+09,9E+09,9E+09,9E+09,9E+09,9E+09]], vmax, z10, tWeldGun;
		ArcLStart [[597.06,-1403.16,-135.36],[0.380481,-0.610502,-0.582596,-0.37829],[-1,0,0,0],[9E+09,9E+09,9E+09,9E+09,9E+09,9E+09]], v50, seam13, weld13\Weave:=weave1, fine, tWeldGun;
		ArcLEnd [[627.18,-1403.07,-135.15],[0.380451,-0.610562,-0.582465,-0.378426],[-1,0,0,0],[9E+09,9E+09,9E+09,9E+09,9E+09,9E+09]], v5, seam13, weld13\Weave:=weave1, fine, tWeldGun;
		MoveL [[628.35,-1412.36,-131.21],[0.467542,-0.524114,-0.539124,-0.464817],[-1,0,0,0],[9E+09,9E+09,9E+09,9E+09,9E+09,9E+09]], vmax, z10, tWeldGun;
		MoveL [[630.04,-1413.39,82.24],[0.406954,-0.557371,-0.567573,-0.448985],[-1,0,0,0],[9E+09,9E+09,9E+09,9E+09,9E+09,9E+09]], vmax, z10, tWeldGun;
		ArcLStart [[626.04,-1395.35,81.99],[0.440579,-0.565277,-0.538288,-0.443394],[-1,0,0,0],[9E+09,9E+09,9E+09,9E+09,9E+09,9E+09]], v40, seam13, weld13\Weave:=weave1, fine, tWeldGun;
		ArcLEnd [[593.22,-1395.33,81.95],[0.440608,-0.565286,-0.538264,-0.443384],[-1,0,0,0],[9E+09,9E+09,9E+09,9E+09,9E+09,9E+09]], v5, seam13, weld13\Weave:=weave1, fine, tWeldGun;
		MoveL [[592.54,-1432.49,82.17],[0.427339,-0.575763,-0.543581,-0.436347],[-1,0,0,0],[9E+09,9E+09,9E+09,9E+09,9E+09,9E+09]], vmax, z10, tWeldGun;
		MoveL [[409.08,-1390.23,81.60],[0.377566,-0.521097,-0.645665,-0.411119],[-1,0,0,0],[9E+09,9E+09,9E+09,9E+09,9E+09,9E+09]], vmax, z10, tWeldGun;
		MoveJ [[483.55,-1400.78,96.25],[0.150969,0.719954,0.110873,0.668268],[-1,0,0,0],[9E+09,9E+09,9E+09,9E+09,9E+09,9E+09]], vmax, z10, tWeldGun;
		MoveL [[586.16,-1400.86,80.98],[0.0313045,0.743014,0.0228137,0.668155],[-1,0,0,0],[9E+09,9E+09,9E+09,9E+09,9E+09,9E+09]], vmax, z10, tWeldGun;
		ArcLStart [[593.68,-1399.47,82.20],[0.0312415,0.743073,0.0227754,0.668093],[-1,0,0,0],[9E+09,9E+09,9E+09,9E+09,9E+09,9E+09]], v50, seam13, weld13\Weave:=weave1, fine, tWeldGun;
		ArcLEnd [[593.72,-1363.60,81.06],[0.0313131,0.743053,0.0226814,0.668115],[-1,0,0,0],[9E+09,9E+09,9E+09,9E+09,9E+09,9E+09]], v5, seam13, weld13\Weave:=weave1, fine, tWeldGun;
		MoveL [[554.18,-1372.28,89.73],[0.15109,0.720146,0.110407,0.668112],[-1,0,0,0],[9E+09,9E+09,9E+09,9E+09,9E+09,9E+09]], vmax, z10, tWeldGun;
		MoveL [[549.71,-1268.25,89.71],[0.151117,0.720151,0.110329,0.668113],[-1,1,0,0],[9E+09,9E+09,9E+09,9E+09,9E+09,9E+09]], vmax, z10, tWeldGun;
		MoveJ [[603.39,-1313.43,143.58],[0.469159,0.533622,-0.523436,0.470269],[-1,-2,3,0],[9E+09,9E+09,9E+09,9E+09,9E+09,9E+09]], vmax, z10, tWeldGun;
		MoveL [[591.28,-1347.97,82.12],[0.473675,0.523571,-0.526883,0.473181],[-1,-2,3,0],[9E+09,9E+09,9E+09,9E+09,9E+09,9E+09]], vmax, z10, tWeldGun;
		ArcLStart [[587.96,-1365.88,81.39],[0.473711,0.523325,-0.527202,0.473062],[-1,-2,3,0],[9E+09,9E+09,9E+09,9E+09,9E+09,9E+09]], v40, seam13, weld13\Weave:=weave1, fine, tWeldGun;
		ArcLEnd [[620.94,-1365.88,81.38],[0.473702,0.523289,-0.527255,0.473052],[-1,-2,3,0],[9E+09,9E+09,9E+09,9E+09,9E+09,9E+09]], v5, seam13, weld13\Weave:=weave1, fine, tWeldGun;
		MoveL [[621.57,-1338.36,83.93],[0.473691,0.523533,-0.526918,0.473168],[-1,-2,3,0],[9E+09,9E+09,9E+09,9E+09,9E+09,9E+09]], vmax, z10, tWeldGun;
		MoveJ [[584.48,-948.55,-60.93],[0.252385,-0.649774,-0.664987,-0.268121],[-1,0,0,0],[9E+09,9E+09,9E+09,9E+09,9E+09,9E+09]], vmax, z10, tWeldGun;
		MoveL [[586.13,-889.04,-107.32],[0.252797,-0.649451,-0.665162,-0.26808],[-1,0,0,0],[9E+09,9E+09,9E+09,9E+09,9E+09,9E+09]], vmax, z10, tWeldGun;
		ArcLStart [[584.57,-887.97,-132.03],[0.253395,-0.649148,-0.665278,-0.267962],[-1,0,0,0],[9E+09,9E+09,9E+09,9E+09,9E+09,9E+09]], v40, seam13, weld13\Weave:=weave1, fine, tWeldGun;
		ArcL [[574.57,-892.86,-134.27],[0.253546,-0.649133,-0.665228,-0.267979],[-1,0,0,0],[9E+09,9E+09,9E+09,9E+09,9E+09,9E+09]], v5, seam13, weld13\Weave:=weave1, z0, tWeldGun;
		ArcL [[475.79,-890.51,-134.53],[0.253539,-0.649165,-0.665195,-0.267991],[-1,0,0,0],[9E+09,9E+09,9E+09,9E+09,9E+09,9E+09]], v5, seam13, weld13\Weave:=weave1, z0, tWeldGun;
		ArcLEnd [[466.55,-879.09,-134.47],[0.253642,-0.649098,-0.665227,-0.267977],[-1,0,0,0],[9E+09,9E+09,9E+09,9E+09,9E+09,9E+09]], v5, seam13, weld13\Weave:=weave1, fine, tWeldGun;
		MoveL [[472.59,-879.09,-111.98],[0.253025,-0.6494,-0.665124,-0.268085],[-1,0,0,0],[9E+09,9E+09,9E+09,9E+09,9E+09,9E+09]], vmax, z10, tWeldGun;
		MoveL [[396.83,-879.33,-105.08],[0.253072,-0.649383,-0.665131,-0.268064],[-1,0,0,0],[9E+09,9E+09,9E+09,9E+09,9E+09,9E+09]], vmax, z10, tWeldGun;
		ArcLStart [[394.25,-876.82,-134.70],[0.258595,-0.647157,-0.667412,-0.262448],[-1,-1,0,0],[9E+09,9E+09,9E+09,9E+09,9E+09,9E+09]], v40, seam13, weld13\Weave:=weave1, fine, tWeldGun;
		ArcL [[381.44,-890.37,-135.06],[0.258791,-0.647168,-0.667273,-0.262579],[-1,-1,0,0],[9E+09,9E+09,9E+09,9E+09,9E+09,9E+09]], v5, seam13, weld13\Weave:=weave1, z0, tWeldGun;
		ArcLEnd [[322.18,-889.35,-135.55],[0.25878,-0.64712,-0.667324,-0.262581],[-1,0,0,0],[9E+09,9E+09,9E+09,9E+09,9E+09,9E+09]], v5, seam13, weld13\Weave:=weave1, fine, tWeldGun;
		MoveL [[322.31,-895.09,-116.44],[0.258649,-0.647181,-0.667323,-0.26256],[-1,0,0,0],[9E+09,9E+09,9E+09,9E+09,9E+09,9E+09]], vmax, z10, tWeldGun;
		MoveL [[273.41,-894.64,-124.57],[0.25314,-0.649501,-0.664982,-0.268082],[-1,0,0,0],[9E+09,9E+09,9E+09,9E+09,9E+09,9E+09]], vmax, z10, tWeldGun;
		ArcLStart [[277.62,-889.74,-135.52],[0.25327,-0.649363,-0.665101,-0.267999],[-1,0,0,0],[9E+09,9E+09,9E+09,9E+09,9E+09,9E+09]], v40, seam13, weld13\Weave:=weave1, fine, tWeldGun;
		ArcLEnd [[220.59,-889.99,-136.94],[0.253257,-0.649434,-0.665002,-0.268085],[-1,0,0,0],[9E+09,9E+09,9E+09,9E+09,9E+09,9E+09]], v5, seam13, weld13\Weave:=weave1, fine, tWeldGun;
		MoveL [[221.58,-928.39,28.18],[0.253244,-0.649506,-0.664879,-0.268227],[-1,0,0,0],[9E+09,9E+09,9E+09,9E+09,9E+09,9E+09]], vmax, z10, tWeldGun;
		MoveL [[149.11,-928.37,24.70],[0.253259,-0.649498,-0.664878,-0.268235],[-1,0,0,0],[9E+09,9E+09,9E+09,9E+09,9E+09,9E+09]], vmax, z10, tWeldGun;
		MoveL [[147.94,-898.55,-125.25],[0.226531,-0.659809,-0.673837,-0.243475],[-1,0,0,0],[9E+09,9E+09,9E+09,9E+09,9E+09,9E+09]], vmax, z10, tWeldGun;
		ArcLStart [[145.94,-889.85,-134.87],[0.226621,-0.659751,-0.673869,-0.243461],[-1,0,0,0],[9E+09,9E+09,9E+09,9E+09,9E+09,9E+09]], v40, seam13, weld13\Weave:=weave1, fine, tWeldGun;
		ArcL [[136.31,-880.56,-133.73],[0.179199,-0.674782,-0.68842,-0.196562],[-1,-1,0,0],[9E+09,9E+09,9E+09,9E+09,9E+09,9E+09]], v5, seam13, weld13\Weave:=weave1, z0, tWeldGun;
		ArcLEnd [[135.53,-866.71,-133.14],[0.179149,-0.674875,-0.688323,-0.196627],[-1,-1,0,0],[9E+09,9E+09,9E+09,9E+09,9E+09,9E+09]], v5, seam13, weld13\Weave:=weave1, fine, tWeldGun;
		MoveL [[135.09,-898.03,-81.67],[0.226532,-0.659739,-0.673982,-0.243263],[-1,0,0,0],[9E+09,9E+09,9E+09,9E+09,9E+09,9E+09]], vmax, z10, tWeldGun;
		MoveJ [[133.84,-1301.69,-30.86],[0.241723,0.664636,-0.669792,0.226294],[-1,-1,-2,0],[9E+09,9E+09,9E+09,9E+09,9E+09,9E+09]], vmax, z10, tWeldGun;
		MoveL [[130.27,-1374.37,-120.54],[0.202113,0.676143,-0.685621,0.178621],[-1,0,-2,0],[9E+09,9E+09,9E+09,9E+09,9E+09,9E+09]], vmax, z10, tWeldGun;
		ArcLStart [[129.21,-1375.14,-130.19],[0.202076,0.676173,-0.685603,0.17862],[-1,0,-2,0],[9E+09,9E+09,9E+09,9E+09,9E+09,9E+09]], v40, seam13, weld13\Weave:=weave1, fine, tWeldGun;
		ArcL [[129.40,-1362.73,-131.77],[0.202045,0.676301,-0.68549,0.178601],[-1,0,-2,0],[9E+09,9E+09,9E+09,9E+09,9E+09,9E+09]], v5, seam13, weld13\Weave:=weave1, z0, tWeldGun;
		ArcLEnd [[141.33,-1351.30,-130.96],[0.202027,0.676304,-0.685497,0.178584],[-1,0,-2,0],[9E+09,9E+09,9E+09,9E+09,9E+09,9E+09]], v5, seam13, weld13\Weave:=weave1, fine, tWeldGun;
		MoveL [[140.84,-1281.82,33.20],[0.241757,0.664658,-0.669788,0.226201],[-1,-1,-2,0],[9E+09,9E+09,9E+09,9E+09,9E+09,9E+09]], vmax, z10, tWeldGun;
		MoveL [[199.15,-1314.71,46.47],[0.241551,0.664904,-0.669698,0.225967],[-1,0,-2,0],[9E+09,9E+09,9E+09,9E+09,9E+09,9E+09]], vmax, z10, tWeldGun;
		MoveL [[212.97,-1340.61,-125.15],[0.241813,0.664699,-0.66974,0.226165],[-1,0,-2,0],[9E+09,9E+09,9E+09,9E+09,9E+09,9E+09]], vmax, z10, tWeldGun;
		ArcLStart [[215.34,-1352.26,-133.17],[0.241825,0.664745,-0.669689,0.226168],[-1,0,-2,0],[9E+09,9E+09,9E+09,9E+09,9E+09,9E+09]], v40, seam13, weld13\Weave:=weave1, fine, tWeldGun;
		ArcLEnd [[270.65,-1353.47,-132.38],[0.241836,0.664718,-0.669712,0.226167],[-1,0,-2,0],[9E+09,9E+09,9E+09,9E+09,9E+09,9E+09]], v5, seam13, weld13\Weave:=weave1, fine, tWeldGun;
		MoveL [[270.66,-1348.41,-112.62],[0.241722,0.664804,-0.669653,0.226213],[-1,0,-2,0],[9E+09,9E+09,9E+09,9E+09,9E+09,9E+09]], vmax, z10, tWeldGun;
		MoveL [[316.82,-1344.16,-112.66],[0.241796,0.664657,-0.669739,0.226309],[-1,0,-2,0],[9E+09,9E+09,9E+09,9E+09,9E+09,9E+09]], vmax, z10, tWeldGun;
		ArcLStart [[315.96,-1353.31,-132.51],[0.241791,0.664741,-0.669685,0.22623],[-1,0,-2,0],[9E+09,9E+09,9E+09,9E+09,9E+09,9E+09]], v40, seam13, weld13\Weave:=weave1, fine, tWeldGun;
		ArcL [[378.49,-1354.48,-133.34],[0.24179,0.664785,-0.669645,0.226217],[-1,0,-2,0],[9E+09,9E+09,9E+09,9E+09,9E+09,9E+09]], v5, seam13, weld13\Weave:=weave1, z0, tWeldGun;
		ArcLEnd [[386.30,-1365.07,-133.55],[0.241806,0.664743,-0.669681,0.226219],[-1,0,-2,0],[9E+09,9E+09,9E+09,9E+09,9E+09,9E+09]], v5, seam13, weld13\Weave:=weave1, fine, tWeldGun;
		MoveL [[388.15,-1371.45,-115.55],[0.241783,0.664794,-0.669629,0.226246],[-1,0,-2,0],[9E+09,9E+09,9E+09,9E+09,9E+09,9E+09]], vmax, z10, tWeldGun;
		MoveL [[460.68,-1363.89,-125.97],[0.241779,0.664811,-0.669612,0.226249],[-1,0,-2,0],[9E+09,9E+09,9E+09,9E+09,9E+09,9E+09]], vmax, z10, tWeldGun;
		ArcLStart [[459.75,-1367.07,-131.60],[0.241795,0.664917,-0.669507,0.226233],[-1,0,-2,0],[9E+09,9E+09,9E+09,9E+09,9E+09,9E+09]], v40, seam13, weld13\Weave:=weave1, fine, tWeldGun;
		ArcL [[471.32,-1354.85,-133.04],[0.241789,0.664914,-0.669523,0.226201],[-1,0,-2,0],[9E+09,9E+09,9E+09,9E+09,9E+09,9E+09]], v5, seam13, weld13\Weave:=weave1, z0, tWeldGun;
		ArcL [[571.50,-1356.03,-133.26],[0.241781,0.664938,-0.669508,0.226183],[-1,0,-2,0],[9E+09,9E+09,9E+09,9E+09,9E+09,9E+09]], v5, seam13, weld13\Weave:=weave1, z0, tWeldGun;
		ArcLEnd [[579.28,-1366.47,-130.48],[0.24184,0.664924,-0.669502,0.226179],[-1,0,-2,0],[9E+09,9E+09,9E+09,9E+09,9E+09,9E+09]], v5, seam13, weld13\Weave:=weave1, fine, tWeldGun;
		MoveL [[580.73,-1359.16,-109.60],[0.211837,0.675037,-0.658293,0.257101],[-1,0,-2,0],[9E+09,9E+09,9E+09,9E+09,9E+09,9E+09]], vmax, z10, tWeldGun;
		MoveL [[580.72,-1333.23,219.73],[0.211837,0.67505,-0.658281,0.257098],[-1,0,-2,0],[9E+09,9E+09,9E+09,9E+09,9E+09,9E+09]], vmax, z10, tWeldGun;
		MoveJ [[285.51,-1411.06,96.42],[0.200981,-0.684372,-0.670688,-0.203517],[-1,-1,0,0],[9E+09,9E+09,9E+09,9E+09,9E+09,9E+09]], vmax, z10, tWeldGun;
		MoveL [[279.17,-1421.93,-119.46],[0.177026,-0.688238,-0.684045,-0.164539],[-1,-1,0,0],[9E+09,9E+09,9E+09,9E+09,9E+09,9E+09]], vmax, z10, tWeldGun;
		ArcLStart [[281.45,-1415.02,-128.28],[0.177385,-0.688168,-0.684016,-0.164566],[-1,-1,0,0],[9E+09,9E+09,9E+09,9E+09,9E+09,9E+09]], v40, seam13, weld13\Weave:=weave1, fine, tWeldGun;
		ArcLEnd [[343.22,-1415.08,-128.29],[0.177414,-0.688148,-0.684031,-0.164558],[-1,-1,0,0],[9E+09,9E+09,9E+09,9E+09,9E+09,9E+09]], v5, seam13, weld13\Weave:=weave1, fine, tWeldGun;
		MoveL [[345.60,-1413.44,-114.91],[0.177186,-0.688241,-0.683983,-0.164611],[-1,-1,0,0],[9E+09,9E+09,9E+09,9E+09,9E+09,9E+09]], vmax, z10, tWeldGun;
		MoveL [[346.28,-1412.31,-127.04],[0.247917,-0.667279,-0.662994,-0.231765],[-1,-1,0,0],[9E+09,9E+09,9E+09,9E+09,9E+09,9E+09]], vmax, z10, tWeldGun;
		ArcLStart [[346.07,-1406.84,-129.30],[0.247993,-0.667283,-0.662971,-0.231741],[-1,-1,0,0],[9E+09,9E+09,9E+09,9E+09,9E+09,9E+09]], v40, seam13, weld13\Weave:=weave1, fine, tWeldGun;
		ArcLEnd [[280.68,-1406.02,-129.12],[0.248008,-0.66729,-0.66296,-0.231735],[-1,-1,0,0],[9E+09,9E+09,9E+09,9E+09,9E+09,9E+09]], v5, seam13, weld13\Weave:=weave1, fine, tWeldGun;
		MoveL [[278.24,-1414.33,-118.08],[0.247841,-0.667243,-0.663091,-0.231675],[-1,-1,0,0],[9E+09,9E+09,9E+09,9E+09,9E+09,9E+09]], vmax, z10, tWeldGun;
		MoveL [[281.30,-1410.99,-125.83],[0.247889,-0.667299,-0.662982,-0.231774],[-1,-1,0,0],[9E+09,9E+09,9E+09,9E+09,9E+09,9E+09]], v200, z10, tWeldGun;
		ArcLStart [[281.21,-1407.29,-131.93],[0.247983,-0.667283,-0.662952,-0.231803],[-1,-1,0,0],[9E+09,9E+09,9E+09,9E+09,9E+09,9E+09]], v40, seam13, weld13\Weave:=weave1, fine, tWeldGun;
		ArcLEnd [[346.15,-1406.93,-131.71],[0.248091,-0.667221,-0.662977,-0.231796],[-1,-1,0,0],[9E+09,9E+09,9E+09,9E+09,9E+09,9E+09]], v5, seam13, weld13\Weave:=weave1, fine, tWeldGun;
		MoveL [[346.31,-1422.77,-122.69],[0.247822,-0.667247,-0.663099,-0.231658],[-1,-1,0,0],[9E+09,9E+09,9E+09,9E+09,9E+09,9E+09]], v200, z10, tWeldGun;
		MoveJ [[748.76,-1435.11,122.90],[0.309636,-0.639534,-0.632199,-0.308944],[-1,0,0,0],[9E+09,9E+09,9E+09,9E+09,9E+09,9E+09]], vmax, z10, tWeldGun;
		MoveL [[713.11,-1431.01,114.74],[0.309534,-0.639554,-0.632247,-0.308909],[-1,0,0,0],[9E+09,9E+09,9E+09,9E+09,9E+09,9E+09]], vmax, z10, tWeldGun;
		ArcLStart [[711.57,-1407.93,114.85],[0.309702,-0.639543,-0.632123,-0.309016],[-1,0,0,0],[9E+09,9E+09,9E+09,9E+09,9E+09,9E+09]], v40, seam13, weld13\Weave:=weave1, fine, tWeldGun;
		ArcLEnd [[692.83,-1407.95,87.57],[0.309767,-0.639507,-0.632187,-0.308892],[-1,0,0,0],[9E+09,9E+09,9E+09,9E+09,9E+09,9E+09]], v5, seam13, weld13\Weave:=weave1, fine, tWeldGun;
		MoveL [[694.62,-1427.85,89.22],[0.309609,-0.639506,-0.63227,-0.308883],[-1,0,0,0],[9E+09,9E+09,9E+09,9E+09,9E+09,9E+09]], v200, z10, tWeldGun;
		MoveL [[713.06,-1431.01,114.71],[0.309564,-0.639548,-0.632251,-0.30888],[-1,0,0,0],[9E+09,9E+09,9E+09,9E+09,9E+09,9E+09]], v200, z10, tWeldGun;
		ArcLStart [[712.95,-1408.22,114.38],[0.309717,-0.639503,-0.632179,-0.308968],[-1,0,0,0],[9E+09,9E+09,9E+09,9E+09,9E+09,9E+09]], v40, seam13, weld13\Weave:=weave1, fine, tWeldGun;
		ArcL [[750.96,-1407.06,114.72],[0.309759,-0.639541,-0.632136,-0.308936],[-1,0,0,0],[9E+09,9E+09,9E+09,9E+09,9E+09,9E+09]], v5, seam13, weld13\Weave:=weave1, z20, tWeldGun;
		ArcL [[757.77,-1407.18,96.42],[0.309876,-0.639582,-0.632001,-0.309009],[-1,0,0,0],[9E+09,9E+09,9E+09,9E+09,9E+09,9E+09]], v5, seam13, weld13\Weave:=weave1, z20, tWeldGun;
		ArcLEnd [[769.81,-1407.71,86.71],[0.309836,-0.639623,-0.63199,-0.308987],[-1,0,0,0],[9E+09,9E+09,9E+09,9E+09,9E+09,9E+09]], v5, seam13, weld13\Weave:=weave1, fine, tWeldGun;
		MoveL [[772.20,-1434.22,91.41],[0.309863,-0.63952,-0.632095,-0.30896],[-1,0,0,0],[9E+09,9E+09,9E+09,9E+09,9E+09,9E+09]], vmax, z10, tWeldGun;
		MoveL [[627.48,-1417.65,-2.71],[0.30978,-0.639664,-0.632044,-0.308849],[-1,0,0,0],[9E+09,9E+09,9E+09,9E+09,9E+09,9E+09]], vmax, z10, tWeldGun;
		ArcLStart [[622.56,-1406.59,-12.22],[0.309929,-0.639535,-0.632206,-0.308635],[-1,0,0,0],[9E+09,9E+09,9E+09,9E+09,9E+09,9E+09]], v40, seam13, weld13\Weave:=weave1, fine, tWeldGun;
		ArcL [[586.80,-1407.81,-64.76],[0.310007,-0.639562,-0.632113,-0.30869],[-1,0,0,0],[9E+09,9E+09,9E+09,9E+09,9E+09,9E+09]], v5, seam13, weld13\Weave:=weave1, z0, tWeldGun;
		ArcLEnd [[547.00,-1408.76,-124.51],[0.310106,-0.639539,-0.632128,-0.308607],[-1,0,0,0],[9E+09,9E+09,9E+09,9E+09,9E+09,9E+09]], v5, seam13, weld13\Weave:=weave1, fine, tWeldGun;
		MoveL [[545.98,-1470.65,-122.68],[0.309529,-0.639772,-0.632153,-0.308653],[-1,0,0,0],[9E+09,9E+09,9E+09,9E+09,9E+09,9E+09]], vmax, z10, tWeldGun;
		MoveL [[546.01,-1470.74,261.49],[0.309463,-0.639811,-0.632171,-0.308601],[-1,0,0,0],[9E+09,9E+09,9E+09,9E+09,9E+09,9E+09]], vmax, z10, tWeldGun;
		MoveJ [[450.72,-1393.79,89.08],[0.00680651,0.918501,-0.0118982,0.395183],[-1,0,-3,0],[9E+09,9E+09,9E+09,9E+09,9E+09,9E+09]], vmax, z10, tWeldGun;
		MoveL [[571.40,-1393.78,20.15],[0.00679519,0.918514,-0.0118615,0.395152],[-1,0,-3,0],[9E+09,9E+09,9E+09,9E+09,9E+09,9E+09]], vmax, z10, tWeldGun;
		ArcLStart [[575.83,-1395.64,7.24],[0.00323578,0.944511,-0.0118289,0.328252],[-1,-1,-3,0],[9E+09,9E+09,9E+09,9E+09,9E+09,9E+09]], v50, seam13, weld13\Weave:=weave1, fine, tWeldGun;
		ArcLEnd [[576.75,-1369.68,7.40],[0.00321436,0.944524,-0.0118118,0.328217],[-1,-1,-3,0],[9E+09,9E+09,9E+09,9E+09,9E+09,9E+09]], v5, seam13, weld13\Weave:=weave1, fine, tWeldGun;
		MoveL [[564.04,-1375.65,36.36],[0.00687019,0.918524,-0.0118557,0.395129],[-1,0,-3,0],[9E+09,9E+09,9E+09,9E+09,9E+09,9E+09]], vmax, z10, tWeldGun;
		MoveJ [[280.70,-816.60,118.66],[0.243228,0.672922,-0.664156,0.216597],[-1,0,-2,0],[9E+09,9E+09,9E+09,9E+09,9E+09,9E+09]], vmax, z10, tWeldGun;
		MoveL [[280.45,-816.02,-119.56],[0.197153,0.688424,-0.669151,0.198599],[-1,0,-2,0],[9E+09,9E+09,9E+09,9E+09,9E+09,9E+09]], vmax, z10, tWeldGun;
		ArcLStart [[280.31,-833.88,-132.23],[0.180282,0.693172,-0.676198,0.172535],[-1,0,-2,0],[9E+09,9E+09,9E+09,9E+09,9E+09,9E+09]], v40, seam13, weld13\Weave:=weave1, fine, tWeldGun;
		ArcLEnd [[342.93,-833.70,-131.64],[0.180266,0.693164,-0.6762,0.172574],[-1,0,-2,0],[9E+09,9E+09,9E+09,9E+09,9E+09,9E+09]], v5, seam13, weld13\Weave:=weave1, fine, tWeldGun;
		MoveL [[342.48,-807.65,-103.06],[0.243058,0.673116,-0.664102,0.216347],[-1,0,-2,0],[9E+09,9E+09,9E+09,9E+09,9E+09,9E+09]], vmax, z10, tWeldGun;
		MoveL [[345.00,-832.65,-129.28],[0.23943,0.676376,-0.664326,0.209427],[-1,0,-2,0],[9E+09,9E+09,9E+09,9E+09,9E+09,9E+09]], vmax, z10, tWeldGun;
		ArcLStart [[344.99,-837.69,-131.04],[0.23944,0.676429,-0.664268,0.209432],[-1,0,-2,0],[9E+09,9E+09,9E+09,9E+09,9E+09,9E+09]], v40, seam13, weld13\Weave:=weave1, fine, tWeldGun;
		ArcLEnd [[279.53,-836.97,-132.08],[0.239403,0.676476,-0.664262,0.20934],[-1,0,-2,0],[9E+09,9E+09,9E+09,9E+09,9E+09,9E+09]], v5, seam13, weld13\Weave:=weave1, fine, tWeldGun;
		MoveL [[282.07,-830.03,-127.27],[0.239368,0.676512,-0.664252,0.209295],[-1,0,-2,0],[9E+09,9E+09,9E+09,9E+09,9E+09,9E+09]], vmax, z10, tWeldGun;
		MoveL [[340.63,-830.01,-127.29],[0.276253,0.663629,-0.647063,0.254147],[-1,-1,-2,0],[9E+09,9E+09,9E+09,9E+09,9E+09,9E+09]], vmax, z10, tWeldGun;
		ArcLStart [[341.79,-839.21,-134.25],[0.276248,0.663637,-0.647056,0.25415],[-1,-1,-2,0],[9E+09,9E+09,9E+09,9E+09,9E+09,9E+09]], v40, seam13, weld13\Weave:=weave1, fine, tWeldGun;
		ArcLEnd [[275.96,-839.30,-134.30],[0.276226,0.663648,-0.647095,0.254046],[-1,-1,-2,0],[9E+09,9E+09,9E+09,9E+09,9E+09,9E+09]], v5, seam13, weld13\Weave:=weave1, fine, tWeldGun;
		MoveL [[278.09,-824.22,-132.32],[0.276187,0.663695,-0.647123,0.253895],[-1,-1,-2,0],[9E+09,9E+09,9E+09,9E+09,9E+09,9E+09]], vmax, z10, tWeldGun;
		MoveL [[714.08,-820.90,116.19],[0.255079,0.669279,-0.660332,0.225751],[-1,0,-2,0],[9E+09,9E+09,9E+09,9E+09,9E+09,9E+09]], vmax, z10, tWeldGun;
		ArcLStart [[711.72,-839.02,114.21],[0.255103,0.669318,-0.660289,0.225732],[-1,0,-2,0],[9E+09,9E+09,9E+09,9E+09,9E+09,9E+09]], v40, seam13, weld13\Weave:=weave1, fine, tWeldGun;
		ArcLEnd [[689.82,-838.03,85.78],[0.255132,0.66942,-0.660194,0.225676],[-1,0,-2,0],[9E+09,9E+09,9E+09,9E+09,9E+09,9E+09]], v5, seam13, weld13\Weave:=weave1, fine, tWeldGun;
		MoveL [[693.54,-821.10,87.96],[0.255102,0.669397,-0.660268,0.225562],[-1,0,-2,0],[9E+09,9E+09,9E+09,9E+09,9E+09,9E+09]], v200, z10, tWeldGun;
		MoveL [[714.11,-820.85,116.18],[0.255054,0.669249,-0.660379,0.225731],[-1,0,-2,0],[9E+09,9E+09,9E+09,9E+09,9E+09,9E+09]], v200, z10, tWeldGun;
		ArcLStart [[712.35,-839.62,114.96],[0.255166,0.669278,-0.660318,0.225695],[-1,0,-2,0],[9E+09,9E+09,9E+09,9E+09,9E+09,9E+09]], v40, seam13, weld13\Weave:=weave1, fine, tWeldGun;
		ArcL [[749.58,-839.57,114.36],[0.255124,0.669325,-0.660279,0.225718],[-1,0,-2,0],[9E+09,9E+09,9E+09,9E+09,9E+09,9E+09]], v5, seam13, weld13\Weave:=weave1, z10, tWeldGun;
		ArcL [[755.54,-839.23,95.73],[0.255123,0.669215,-0.66041,0.225659],[-1,0,-2,0],[9E+09,9E+09,9E+09,9E+09,9E+09,9E+09]], v5, seam13, weld13\Weave:=weave1, z10, tWeldGun;
		ArcLEnd [[767.76,-839.65,85.57],[0.255158,0.669169,-0.660424,0.225719],[-1,0,-2,0],[9E+09,9E+09,9E+09,9E+09,9E+09,9E+09]], v5, seam13, weld13\Weave:=weave1, fine, tWeldGun;
		MoveL [[772.08,-767.27,86.77],[0.255103,0.66918,-0.660433,0.225721],[-1,0,-2,0],[9E+09,9E+09,9E+09,9E+09,9E+09,9E+09]], vmax, z10, tWeldGun;
		MoveL [[627.18,-826.93,-5.83],[0.253508,0.65756,-0.66005,0.26016],[-1,0,-2,0],[9E+09,9E+09,9E+09,9E+09,9E+09,9E+09]], vmax, z10, tWeldGun;
		ArcLStart [[625.59,-838.29,-9.60],[0.253597,0.657512,-0.659967,0.260404],[-1,0,-2,0],[9E+09,9E+09,9E+09,9E+09,9E+09,9E+09]], v40, seam13, weld13\Weave:=weave1, fine, tWeldGun;
		ArcL [[579.59,-838.82,-74.40],[0.253602,0.657534,-0.659951,0.260383],[-1,0,-2,0],[9E+09,9E+09,9E+09,9E+09,9E+09,9E+09]], v5, seam13, weld13\Weave:=weave1, z0, tWeldGun;
		ArcLEnd [[541.11,-838.82,-130.24],[0.253635,0.657488,-0.659927,0.260529],[-1,0,-2,0],[9E+09,9E+09,9E+09,9E+09,9E+09,9E+09]], v5, seam13, weld13\Weave:=weave1, fine, tWeldGun;
		MoveL [[548.88,-773.40,234.33],[0.243177,0.673515,-0.663846,0.215757],[-1,0,-2,0],[9E+09,9E+09,9E+09,9E+09,9E+09,9E+09]], vmax, z10, tWeldGun;
		MoveJ [[554.61,-845.95,234.31],[0.0125503,-0.913958,0.00705174,-0.405554],[-1,0,-3,0],[9E+09,9E+09,9E+09,9E+09,9E+09,9E+09]], vmax, z10, tWeldGun;
		MoveL [[577.03,-856.78,17.59],[0.00389083,-0.924944,0.010701,-0.379933],[-1,-1,-3,0],[9E+09,9E+09,9E+09,9E+09,9E+09,9E+09]], vmax, z10, tWeldGun;
		ArcLStart [[581.29,-855.54,4.69],[0.00394985,-0.924973,0.0105669,-0.379867],[-1,-1,-3,0],[9E+09,9E+09,9E+09,9E+09,9E+09,9E+09]], v40, seam13, weld13\Weave:=weave1, fine, tWeldGun;
		ArcLEnd [[581.36,-879.94,4.55],[0.00400335,-0.924982,0.0105343,-0.379844],[-1,-1,-3,0],[9E+09,9E+09,9E+09,9E+09,9E+09,9E+09]], v5, seam13, weld13\Weave:=weave1, fine, tWeldGun;
		MoveL [[536.09,-886.10,63.12],[0.0125865,-0.913974,0.00698526,-0.405519],[-1,0,-3,0],[9E+09,9E+09,9E+09,9E+09,9E+09,9E+09]], vmax, z10, tWeldGun;
		MoveJ [[471.77,-923.60,234.81],[0.361351,0.15882,-0.917288,0.0527665],[-1,0,-1,0],[9E+09,9E+09,9E+09,9E+09,9E+09,9E+09]], vmax, z10, tWeldGun;
		MoveL [[900.49,-837.79,215.66],[0.339396,0.215461,-0.903746,0.147074],[-1,-1,-1,0],[9E+09,9E+09,9E+09,9E+09,9E+09,9E+09]], vmax, z10, tWeldGun;
		MoveL [[900.44,-837.75,127.43],[0.339421,0.215477,-0.903738,0.147042],[-1,-1,-1,0],[9E+09,9E+09,9E+09,9E+09,9E+09,9E+09]], vmax, z10, tWeldGun;
		ArcLStart [[891.28,-846.19,116.68],[0.339399,0.215507,-0.90374,0.147034],[-1,-1,-1,0],[9E+09,9E+09,9E+09,9E+09,9E+09,9E+09]], v40, seam13, weld13\Weave:=weave1, fine, tWeldGun;
		ArcLEnd [[890.65,-846.37,81.46],[0.339418,0.215511,-0.903735,0.147018],[-1,-1,-1,0],[9E+09,9E+09,9E+09,9E+09,9E+09,9E+09]], v5, seam13, weld13\Weave:=weave1, fine, tWeldGun;
		MoveL [[900.41,-837.71,81.46],[0.339442,0.215511,-0.903726,0.147016],[-1,-1,-1,0],[9E+09,9E+09,9E+09,9E+09,9E+09,9E+09]], vmax, z10, tWeldGun;
		MoveL [[900.39,-837.71,198.80],[0.339465,0.215526,-0.903715,0.147012],[-1,-1,-1,0],[9E+09,9E+09,9E+09,9E+09,9E+09,9E+09]], vmax, z10, tWeldGun;
		MoveJ [[893.27,-898.66,198.53],[0.473399,-0.27429,-0.79444,-0.263675],[-1,0,-1,0],[9E+09,9E+09,9E+09,9E+09,9E+09,9E+09]], vmax, z10, tWeldGun;
		MoveL [[893.26,-898.66,124.83],[0.4734,-0.274289,-0.794437,-0.263683],[-1,0,-1,0],[9E+09,9E+09,9E+09,9E+09,9E+09,9E+09]], vmax, z10, tWeldGun;
		ArcLStart [[887.28,-891.68,117.80],[0.48296,-0.257091,-0.803409,-0.234924],[-1,0,-1,0],[9E+09,9E+09,9E+09,9E+09,9E+09,9E+09]], v40, seam13, weld13\Weave:=weave1, fine, tWeldGun;
		ArcLEnd [[887.29,-891.67,77.79],[0.477055,-0.267897,-0.797911,-0.25296],[-1,0,-1,0],[9E+09,9E+09,9E+09,9E+09,9E+09,9E+09]], v5, seam13, weld13\Weave:=weave1, fine, tWeldGun;
		MoveL [[937.32,-934.77,92.77],[0.477007,-0.267909,-0.797948,-0.252921],[-1,0,-1,0],[9E+09,9E+09,9E+09,9E+09,9E+09,9E+09]], vmax, z10, tWeldGun;
		MoveL [[898.69,-1405.03,162.74],[0.405782,-0.372754,-0.813112,-0.187737],[-1,-1,-1,0],[9E+09,9E+09,9E+09,9E+09,9E+09,9E+09]], vmax, z10, tWeldGun;
		MoveL [[893.71,-1403.99,128.70],[0.405776,-0.37274,-0.81311,-0.187787],[-1,-1,-1,0],[9E+09,9E+09,9E+09,9E+09,9E+09,9E+09]], vmax, z10, tWeldGun;
		ArcLStart [[884.67,-1404.01,118.73],[0.405809,-0.372745,-0.8131,-0.187747],[-1,-1,-1,0],[9E+09,9E+09,9E+09,9E+09,9E+09,9E+09]], v40, seam13, weld13\Weave:=weave1, fine, tWeldGun;
		ArcLEnd [[884.66,-1404.02,87.70],[0.40582,-0.372749,-0.813094,-0.187742],[-1,-1,-1,0],[9E+09,9E+09,9E+09,9E+09,9E+09,9E+09]], v5, seam13, weld13\Weave:=weave1, fine, tWeldGun;
		MoveL [[899.80,-1417.41,147.01],[0.405769,-0.372778,-0.81311,-0.187726],[-1,-1,-1,0],[9E+09,9E+09,9E+09,9E+09,9E+09,9E+09]], vmax, z10, tWeldGun;
		MoveJ [[891.04,-1353.86,172.64],[0.459453,0.258247,-0.822177,0.215029],[-1,-1,-1,0],[9E+09,9E+09,9E+09,9E+09,9E+09,9E+09]], vmax, z10, tWeldGun;
		MoveL [[890.95,-1353.84,123.85],[0.45951,0.258257,-0.822151,0.214995],[-1,-1,-1,0],[9E+09,9E+09,9E+09,9E+09,9E+09,9E+09]], vmax, z10, tWeldGun;
		ArcLStart [[883.98,-1356.19,118.84],[0.459511,0.258226,-0.822164,0.214982],[-1,-1,-1,0],[9E+09,9E+09,9E+09,9E+09,9E+09,9E+09]], v40, seam13, weld13\Weave:=weave1, fine, tWeldGun;
		ArcLEnd [[883.33,-1356.75,82.88],[0.459529,0.258231,-0.822154,0.214972],[-1,-1,-1,0],[9E+09,9E+09,9E+09,9E+09,9E+09,9E+09]], v5, seam13, weld13\Weave:=weave1, fine, tWeldGun;
		MoveL [[954.45,-1305.33,82.88],[0.459526,0.258233,-0.822153,0.21498],[-1,-1,-1,0],[9E+09,9E+09,9E+09,9E+09,9E+09,9E+09]], vmax, z10, tWeldGun;
		MoveL [[954.64,-1305.47,331.71],[0.459382,0.258257,-0.822177,0.215165],[-1,-1,-1,0],[9E+09,9E+09,9E+09,9E+09,9E+09,9E+09]], vmax, z10, tWeldGun;
		MoveJ [[785.08,-1364.00,203.32],[0.00171317,-0.947718,0.00701896,-0.319029],[-1,-1,1,0],[9E+09,9E+09,9E+09,9E+09,9E+09,9E+09]], vmax, z10, tWeldGun;
		MoveL [[803.47,-1368.09,131.07],[0.00412255,-0.937659,0.00608177,-0.347481],[-1,-1,1,0],[9E+09,9E+09,9E+09,9E+09,9E+09,9E+09]], vmax, z10, tWeldGun;
		ArcLStart [[804.13,-1366.42,123.85],[0.00419124,-0.937702,0.00597678,-0.347365],[-1,-1,1,0],[9E+09,9E+09,9E+09,9E+09,9E+09,9E+09]], v40, seam13, weld13\Weave:=weave1, fine, tWeldGun;
		ArcLEnd [[804.13,-1396.73,123.94],[0.00421357,-0.937701,0.00598234,-0.347367],[-1,-1,1,0],[9E+09,9E+09,9E+09,9E+09,9E+09,9E+09]], v5, seam13, weld13\Weave:=weave1, fine, tWeldGun;
		MoveL [[799.72,-1397.77,160.94],[0.00406041,-0.937645,0.00597838,-0.34752],[-1,-1,1,0],[9E+09,9E+09,9E+09,9E+09,9E+09,9E+09]], vmax, z10, tWeldGun;
		MoveJ [[912.45,-910.97,281.24],[0.471963,-0.00834501,-0.88125,-0.0240746],[-1,-1,-1,0],[9E+09,9E+09,9E+09,9E+09,9E+09,9E+09]], vmax, z10, tWeldGun;
		MoveL [[909.26,-887.50,143.89],[0.306131,-0.0105667,-0.951842,-0.0130303],[-1,0,-1,0],[9E+09,9E+09,9E+09,9E+09,9E+09,9E+09]], vmax, z10, tWeldGun;
		ArcLStart [[895.38,-884.91,123.01],[0.306206,-0.0106151,-0.951816,-0.0131321],[-1,0,-1,0],[9E+09,9E+09,9E+09,9E+09,9E+09,9E+09]], v40, seam13, weld13\Weave:=weave1, fine, tWeldGun;
		ArcLEnd [[895.62,-855.31,122.99],[0.306213,-0.0106343,-0.951813,-0.0131465],[-1,0,-1,0],[9E+09,9E+09,9E+09,9E+09,9E+09,9E+09]], v5, seam13, weld13\Weave:=weave1, fine, tWeldGun;
		MoveL [[912.81,-855.15,147.89],[0.30614,-0.0105141,-0.95184,-0.0129908],[-1,0,-1,0],[9E+09,9E+09,9E+09,9E+09,9E+09,9E+09]], vmax, z10, tWeldGun;
		MoveJ [[902.72,-1362.89,137.84],[0.306146,-0.0105253,-0.951838,-0.0129664],[-1,0,-1,0],[9E+09,9E+09,9E+09,9E+09,9E+09,9E+09]], vmax, z10, tWeldGun;
		MoveL [[908.97,-1368.68,133.52],[0.305903,-0.0107467,-0.951921,-0.0124571],[-1,0,-1,0],[9E+09,9E+09,9E+09,9E+09,9E+09,9E+09]], vmax, z10, tWeldGun;
		ArcLStart [[891.85,-1362.07,124.85],[0.305985,-0.010764,-0.951893,-0.0125866],[-1,0,-1,0],[9E+09,9E+09,9E+09,9E+09,9E+09,9E+09]], v40, seam13, weld13\Weave:=weave1, fine, tWeldGun;
		ArcLEnd [[891.60,-1393.64,124.58],[0.306016,-0.0107572,-0.951883,-0.0125206],[-1,0,-1,0],[9E+09,9E+09,9E+09,9E+09,9E+09,9E+09]], v5, seam13, weld13\Weave:=weave1, fine, tWeldGun;
		MoveL [[900.37,-1394.95,165.72],[0.306084,-0.0106333,-0.95186,-0.0127431],[-1,0,-1,0],[9E+09,9E+09,9E+09,9E+09,9E+09,9E+09]], vmax, z10, tWeldGun;
		MoveJ [[778.65,-875.76,193.58],[0.0091964,-0.885136,-0.0131126,-0.465058],[-1,0,1,0],[9E+09,9E+09,9E+09,9E+09,9E+09,9E+09]], vmax, z10, tWeldGun;
		MoveL [[804.53,-888.57,142.41],[0.00795263,-0.941332,-0.0147738,-0.337067],[-1,-1,1,0],[9E+09,9E+09,9E+09,9E+09,9E+09,9E+09]], vmax, z10, tWeldGun;
		ArcLStart [[807.14,-888.84,121.83],[0.0115328,-0.957016,-0.0172521,-0.289293],[-1,-1,1,0],[9E+09,9E+09,9E+09,9E+09,9E+09,9E+09]], v40, seam13, weld13\Weave:=weave1, fine, tWeldGun;
		ArcLEnd [[807.38,-858.36,122.23],[0.0115657,-0.956979,-0.0171252,-0.289422],[-1,-1,1,0],[9E+09,9E+09,9E+09,9E+09,9E+09,9E+09]], v5, seam13, weld13\Weave:=weave1, fine, tWeldGun;
		MoveL [[808.29,-857.12,184.20],[0.00793204,-0.941309,-0.0148666,-0.337126],[-1,-1,1,0],[9E+09,9E+09,9E+09,9E+09,9E+09,9E+09]], vmax, z10, tWeldGun;
		MoveJ [[948.68,-756.38,498.60],[0.0965323,0.230115,0.963612,0.0958222],[-1,0,3,0],[9E+09,9E+09,9E+09,9E+09,9E+09,9E+09]], vmax, z10, tWeldGun;
		MoveJ [[-77.16,-639.19,851.16],[0.250005,-0.698591,-0.608804,-0.280759],[-2,-1,4,0],[9E+09,9E+09,9E+09,9E+09,9E+09,9E+09]], vmax, z10, tWeldGun;
	ENDPROC
	PROC rRUNSide1A()
           	rTestPosTop;
		TPWrite "Side 1 A";
		MoveJ pSafeS1, vmax, fine, tWeldGun;
		!Code Goes Here
		MoveJ [[1195.77,967.47,624.34],[0.0211986,-0.292543,0.866333,0.404273],[0,-1,1,1],[9E+09,9E+09,9E+09,9E+09,9E+09,9E+09]], v1000, z20, tWeldGun;
		MoveJ [[1202.08,958.55,27.66],[0.0678226,-0.111826,0.895436,0.425548],[0,-1,0,1],[9E+09,9E+09,9E+09,9E+09,9E+09,9E+09]], v1000, z20, tWeldGun;
		!SingArea\Wrist;
		MoveL [[1208.05,954.10,0.64],[0.135152,-0.0819873,0.912838,0.376484],[0,0,0,1],[9E+09,9E+09,9E+09,9E+09,9E+09,9E+09]], v1000, z5, tWeldGun;
		ArcLStart [[1211.29,968.27,-0.59],[0.136515,-0.0793352,0.919743,0.359364],[0,0,0,1],[9E+09,9E+09,9E+09,9E+09,9E+09,9E+09]], v30, seam13, weld13\Weave:=weave1, fine, tWeldGun;
		ArcLEnd [[1181.88,968.48,-1.21],[0.136499,-0.079344,0.919744,0.359366],[0,0,0,1],[9E+09,9E+09,9E+09,9E+09,9E+09,9E+09]], v5, seam13, weld13\Weave:=weave1, fine, tWeldGun;
		MoveL [[1180.50,960.73,100.66],[0.067842,-0.111808,0.895423,0.425576],[0,-1,0,1],[9E+09,9E+09,9E+09,9E+09,9E+09,9E+09]], vmax, z0, tWeldGun;
		MoveL [[867.04,1014.85,67.84],[0.0692843,-0.0563275,0.92497,-0.369403],[0,1,-1,1],[9E+09,9E+09,9E+09,9E+09,9E+09,9E+09]], vmax, z0, tWeldGun;
		MoveL [[869.49,1011.42,-5.10],[0.0692967,-0.0563794,0.924948,-0.369448],[0,1,-1,1],[9E+09,9E+09,9E+09,9E+09,9E+09,9E+09]], vmax, z0, tWeldGun;
		ArcLStart [[870.23,1004.64,-6.00],[0.0692199,-0.0564569,0.924914,-0.369535],[0,1,-1,1],[9E+09,9E+09,9E+09,9E+09,9E+09,9E+09]], v30, seam13, weld13\Weave:=weave1, fine, tWeldGun;
		ArcLEnd [[893.80,1004.78,-6.05],[0.0692111,-0.0564445,0.92492,-0.369524],[0,1,-1,1],[9E+09,9E+09,9E+09,9E+09,9E+09,9E+09]], v5, seam13, weld13\Weave:=weave1, fine, tWeldGun;
		MoveL [[886.66,1008.91,119.93],[0.0693309,-0.056349,0.924962,-0.369411],[0,1,-1,1],[9E+09,9E+09,9E+09,9E+09,9E+09,9E+09]], vmax, z0, tWeldGun;
		MoveL [[1179.30,1008.46,86.74],[0.107531,-0.15675,0.912414,-0.362448],[0,0,-1,1],[9E+09,9E+09,9E+09,9E+09,9E+09,9E+09]], vmax, z0, tWeldGun;
		MoveL [[1183.28,1011.87,-7.09],[0.107529,-0.156762,0.912406,-0.362464],[0,0,-1,1],[9E+09,9E+09,9E+09,9E+09,9E+09,9E+09]], vmax, z0, tWeldGun;
		ArcLStart [[1182.50,1009.08,-6.44],[0.107436,-0.156815,0.91237,-0.362557],[0,0,-1,1],[9E+09,9E+09,9E+09,9E+09,9E+09,9E+09]], v30, seam13, weld13\Weave:=weave1, fine, tWeldGun;
		ArcLEnd [[1213.91,1008.43,-6.46],[0.107447,-0.156842,0.912362,-0.362564],[0,0,-1,1],[9E+09,9E+09,9E+09,9E+09,9E+09,9E+09]], v5, seam13, weld13\Weave:=weave1, fine, tWeldGun;
		MoveL [[1201.36,1025.64,129.06],[0.213207,-0.193181,0.897428,-0.334435],[0,0,-1,1],[9E+09,9E+09,9E+09,9E+09,9E+09,9E+09]], vmax, z0, tWeldGun;
		MoveJ [[885.83,967.12,146.79],[0.0390937,-0.243498,0.889932,0.383668],[0,-1,0,1],[9E+09,9E+09,9E+09,9E+09,9E+09,9E+09]], vmax, z0, tWeldGun;
		MoveL [[894.90,956.27,69.85],[0.0870766,0.0253294,0.943056,0.320035],[0,0,0,1],[9E+09,9E+09,9E+09,9E+09,9E+09,9E+09]], vmax, z0, tWeldGun;
		MoveL [[897.77,955.06,6.57],[0.0949838,0.0234038,0.90292,0.418528],[0,0,0,1],[9E+09,9E+09,9E+09,9E+09,9E+09,9E+09]], vmax, z0, tWeldGun;
		ArcLStart [[897.02,965.79,-1.05],[0.0949391,0.0234364,0.902969,0.418431],[0,0,0,1],[9E+09,9E+09,9E+09,9E+09,9E+09,9E+09]], v30, seam13, weld13\Weave:=weave1, fine, tWeldGun;
		ArcLEnd [[868.02,967.05,-2.12],[0.0928062,0.0262205,0.917307,0.386327],[0,0,0,1],[9E+09,9E+09,9E+09,9E+09,9E+09,9E+09]], v5, seam13, weld13\Weave:=weave1, fine, tWeldGun;
		MoveL [[862.21,949.49,214.06],[0.0424258,-0.242958,0.89504,0.371585],[0,-1,0,1],[9E+09,9E+09,9E+09,9E+09,9E+09,9E+09]], vmax, z0, tWeldGun;
		MoveL [[1197.39,1502.39,137.74],[0.0213351,-0.292247,0.866338,0.404469],[0,-1,0,1],[9E+09,9E+09,9E+09,9E+09,9E+09,9E+09]], vmax, z0, tWeldGun;
		MoveL [[1212.43,1503.61,12.77],[0.123742,-0.0547004,0.912363,0.386381],[0,0,0,1],[9E+09,9E+09,9E+09,9E+09,9E+09,9E+09]], vmax, z0, tWeldGun;
		ArcLStart [[1212.49,1515.21,0.73],[0.123687,-0.0547013,0.912376,0.386367],[0,0,0,1],[9E+09,9E+09,9E+09,9E+09,9E+09,9E+09]], v30, seam13, weld13\Weave:=weave1, fine, tWeldGun;
		ArcLEnd [[1185.29,1515.16,0.46],[0.123682,-0.0546805,0.912389,0.386341],[0,0,0,1],[9E+09,9E+09,9E+09,9E+09,9E+09,9E+09]], v5, seam13, weld13\Weave:=weave1, fine, tWeldGun;
		MoveL [[1181.48,1503.16,158.48],[0.0212657,-0.292228,0.86634,0.404483],[0,-1,0,1],[9E+09,9E+09,9E+09,9E+09,9E+09,9E+09]], vmax, z0, tWeldGun;
		SingArea\Wrist;
		MoveL [[868.25,1555.51,187.44],[0.227112,-0.185081,0.888817,-0.352378],[0,1,-2,1],[9E+09,9E+09,9E+09,9E+09,9E+09,9E+09]], vmax, z0, tWeldGun;
		MoveL [[868.98,1562.79,2.00],[0.0827412,0.288792,-0.895538,0.328277],[0,1,-2,1],[9E+09,9E+09,9E+09,9E+09,9E+09,9E+09]], vmax, z0, tWeldGun;
		ArcLStart [[868.80,1557.80,-10.94],[0.0827537,0.288837,-0.895507,0.328318],[0,1,-2,1],[9E+09,9E+09,9E+09,9E+09,9E+09,9E+09]], v40, seam13, weld13\Weave:=weave1, fine, tWeldGun;
		ArcLEnd [[890.47,1557.45,-10.78],[0.0827822,0.288828,-0.895499,0.328341],[0,1,-2,1],[9E+09,9E+09,9E+09,9E+09,9E+09,9E+09]], v5, seam13, weld13\Weave:=weave1, fine, tWeldGun;
		MoveL [[888.12,1562.49,80.36],[0.227116,-0.185107,0.888791,-0.352426],[0,1,-2,1],[9E+09,9E+09,9E+09,9E+09,9E+09,9E+09]], vmax, z0, tWeldGun;
		MoveL [[1184.50,1555.09,41.59],[0.152145,-0.176338,0.927538,-0.292285],[0,1,-2,1],[9E+09,9E+09,9E+09,9E+09,9E+09,9E+09]], vmax, z0, tWeldGun;
		MoveL [[1177.05,1568.70,-9.93],[0.112232,0.626696,-0.699388,0.32483],[0,1,-3,1],[9E+09,9E+09,9E+09,9E+09,9E+09,9E+09]], vmax, z0, tWeldGun;
		ArcLStart [[1176.95,1563.04,-11.76],[0.112349,0.626693,-0.699392,0.324785],[0,1,-3,1],[9E+09,9E+09,9E+09,9E+09,9E+09,9E+09]], v30, seam13, weld13\Weave:=weave1, fine, tWeldGun;
		ArcLEnd [[1201.31,1562.19,-12.75],[0.112369,0.626691,-0.699389,0.32479],[0,1,-3,1],[9E+09,9E+09,9E+09,9E+09,9E+09,9E+09]], v5, seam13, weld13\Weave:=weave1, fine, tWeldGun;
		MoveL [[1205.97,1566.31,170.25],[0.227077,-0.185152,0.88879,-0.352432],[0,0,-2,1],[9E+09,9E+09,9E+09,9E+09,9E+09,9E+09]], vmax, z0, tWeldGun;
		MoveL [[881.77,1504.38,147.85],[0.0212859,-0.292306,0.866337,0.404431],[0,-1,0,1],[9E+09,9E+09,9E+09,9E+09,9E+09,9E+09]], vmax, z0, tWeldGun;
		MoveL [[868.22,1500.18,5.30],[0.0257172,0.126447,0.911081,0.391513],[0,0,0,1],[9E+09,9E+09,9E+09,9E+09,9E+09,9E+09]], vmax, z0, tWeldGun;
		ArcLStart [[868.71,1511.36,-5.52],[0.0255875,0.126486,0.911104,0.391455],[0,0,0,1],[9E+09,9E+09,9E+09,9E+09,9E+09,9E+09]], v30, seam13, weld13\Weave:=weave1, fine, tWeldGun;
		ArcLEnd [[894.77,1511.39,-5.46],[0.0256421,0.1265,0.911082,0.391498],[0,0,0,1],[9E+09,9E+09,9E+09,9E+09,9E+09,9E+09]], v5, seam13, weld13\Weave:=weave1, fine, tWeldGun;
		MoveL [[865.68,1505.22,88.67],[0.0212437,-0.292287,0.866358,0.404403],[0,-1,0,1],[9E+09,9E+09,9E+09,9E+09,9E+09,9E+09]], vmax, z0, tWeldGun;
		MoveL [[42.29,1547.28,5.42],[0.0930027,-0.145662,0.911404,0.373466],[1,0,0,1],[9E+09,9E+09,9E+09,9E+09,9E+09,9E+09]], vmax, z0, tWeldGun;
		ArcLStart [[44.93,1558.27,-2.62],[0.0927871,-0.145552,0.911443,0.373466],[1,0,0,1],[9E+09,9E+09,9E+09,9E+09,9E+09,9E+09]], v30, seam13, weld13\Weave:=weave1, fine, tWeldGun;
		ArcLEnd [[10.75,1558.26,-2.66],[0.0927428,-0.145507,0.911453,0.373472],[1,0,0,1],[9E+09,9E+09,9E+09,9E+09,9E+09,9E+09]], v5, seam13, weld13\Weave:=weave1, fine, tWeldGun;
		MoveL [[12.10,1550.46,9.38],[0.0929989,-0.14565,0.911414,0.373447],[1,0,0,1],[9E+09,9E+09,9E+09,9E+09,9E+09,9E+09]], vmax, z0, tWeldGun;
		MoveL [[-278.66,1557.62,11.31],[0.104661,-0.181311,0.91043,0.356779],[1,0,0,1],[9E+09,9E+09,9E+09,9E+09,9E+09,9E+09]], vmax, z0, tWeldGun;
		ArcLStart [[-274.61,1561.39,-0.57],[0.104618,-0.18131,0.910431,0.356787],[1,0,0,1],[9E+09,9E+09,9E+09,9E+09,9E+09,9E+09]], v30, seam13, weld13\Weave:=weave1, fine, tWeldGun;
		ArcLEnd [[-307.86,1561.47,-0.56],[0.104645,-0.181388,0.910415,0.356782],[1,0,0,1],[9E+09,9E+09,9E+09,9E+09,9E+09,9E+09]], v5, seam13, weld13\Weave:=weave1, fine, tWeldGun;
		MoveL [[-319.66,1562.55,534.71],[0.0907184,-0.623281,0.712938,0.30824],[1,0,0,1],[9E+09,9E+09,9E+09,9E+09,9E+09,9E+09]], vmax, z0, tWeldGun;
		MoveJ [[-204.06,743.62,410.35],[0.169831,0.702229,0.669586,-0.1723],[1,0,-2,0],[9E+09,9E+09,9E+09,9E+09,9E+09,9E+09]], vmax, z0, tWeldGun;
		MoveJ [[-336.86,555.26,14.49],[0.352891,0.90921,0.19794,-0.0981131],[0,0,-2,0],[9E+09,9E+09,9E+09,9E+09,9E+09,9E+09]], vmax, z0, tWeldGun;
		ArcLStart [[-338.00,546.88,7.96],[0.35293,0.90919,0.197978,-0.0980772],[0,0,-2,0],[9E+09,9E+09,9E+09,9E+09,9E+09,9E+09]], v30, seam13, weld13\Weave:=weave1, fine, tWeldGun;
		ArcLEnd [[-305.97,545.83,7.77],[0.352984,0.909169,0.197976,-0.0980787],[0,0,-2,0],[9E+09,9E+09,9E+09,9E+09,9E+09,9E+09]], v5, seam13, weld13\Weave:=weave1, fine, tWeldGun;
		MoveL [[-306.62,555.42,20.36],[0.352823,0.909224,0.197986,-0.0981282],[0,0,-2,0],[9E+09,9E+09,9E+09,9E+09,9E+09,9E+09]], vmax, z0, tWeldGun;
		MoveL [[-15.36,553.36,14.76],[0.325268,0.908092,0.244403,-0.0991795],[0,0,-2,0],[9E+09,9E+09,9E+09,9E+09,9E+09,9E+09]], vmax, z0, tWeldGun;
		ArcLStart [[-17.82,544.50,7.92],[0.325299,0.908093,0.244374,-0.0991441],[0,0,-2,0],[9E+09,9E+09,9E+09,9E+09,9E+09,9E+09]], v30, seam13, weld13\Weave:=weave1, fine, tWeldGun;
		ArcLEnd [[12.80,543.57,6.91],[0.325307,0.90808,0.24441,-0.0991463],[0,0,-2,0],[9E+09,9E+09,9E+09,9E+09,9E+09,9E+09]], v5, seam13, weld13\Weave:=weave1, fine, tWeldGun;
		MoveL [[16.53,551.56,14.73],[0.325268,0.908096,0.244389,-0.0991872],[0,0,-2,0],[9E+09,9E+09,9E+09,9E+09,9E+09,9E+09]], vmax, z0, tWeldGun;
		MoveL [[835.19,546.59,8.86],[0.354374,0.887507,0.294518,0.00309851],[0,-1,-2,0],[9E+09,9E+09,9E+09,9E+09,9E+09,9E+09]], vmax, z0, tWeldGun;
		ArcLStart [[835.40,539.24,2.84],[0.354384,0.887506,0.294511,0.00300171],[0,-1,-2,0],[9E+09,9E+09,9E+09,9E+09,9E+09,9E+09]], v30, seam13, weld13\Weave:=weave1, fine, tWeldGun;
		ArcLEnd [[864.16,539.26,2.03],[0.354392,0.887509,0.294492,0.002972],[0,-1,-2,0],[9E+09,9E+09,9E+09,9E+09,9E+09,9E+09]], v5, seam13, weld13\Weave:=weave1, fine, tWeldGun;
		MoveL [[863.15,544.60,13.06],[0.354372,0.887507,0.29452,0.00310136],[0,-1,-2,0],[9E+09,9E+09,9E+09,9E+09,9E+09,9E+09]], vmax, z0, tWeldGun;
		ConfL\Off;
		MoveL [[1163.05,540.25,17.31],[0.272611,0.697866,0.657915,-0.0762502],[0,-1,-3,0],[9E+09,9E+09,9E+09,9E+09,9E+09,9E+09]], vmax, z0, tWeldGun;
		ArcLStart [[1166.60,534.26,6.34],[0.272593,0.697855,0.657923,-0.0763491],[0,-1,-3,0],[9E+09,9E+09,9E+09,9E+09,9E+09,9E+09]], v30, seam13, weld13\Weave:=weave1, fine, tWeldGun;
		ArcLEnd [[1195.65,534.51,5.72],[0.272623,0.697857,0.657916,-0.0762825],[0,-1,-3,0],[9E+09,9E+09,9E+09,9E+09,9E+09,9E+09]], v5, seam13, weld13\Weave:=weave1, fine, tWeldGun;
		MoveL [[1196.79,537.72,478.96],[0.266966,0.671404,0.686159,-0.0844522],[0,-1,-3,0],[9E+09,9E+09,9E+09,9E+09,9E+09,9E+09]], vmax, z10, tWeldGun;
		!MoveJ [[44.07,948.69,1172.83],[0.0459633,-0.688402,0.722614,0.0426485],[0,-1,0,0],[9E+09,9E+09,9E+09,9E+09,9E+09,9E+09]], vmax, z10, tWeldGun;
		MoveJ [[-340.94,933.57,290.70],[0.111592,-0.946666,-0.184924,-0.23911],[1,0,-2,0],[9E+09,9E+09,9E+09,9E+09,9E+09,9E+09]], vmax, z10, tWeldGun;
		MoveL [[-397.78,986.25,11.78],[0.351596,0.0366706,-0.934077,-0.0503611],[1,-1,-3,0],[9E+09,9E+09,9E+09,9E+09,9E+09,9E+09]], v1000, z1, tWeldGun;
		ArcLStart [[-401.31,985.79,-8.73],[0.351547,0.0366966,-0.934101,-0.0502319],[1,-1,-3,0],[9E+09,9E+09,9E+09,9E+09,9E+09,9E+09]], v30, seam13, weld13\Weave:=weave1, fine, tWeldGun;
		ArcL [[-401.70,963.07,-8.24],[0.351611,0.0366522,-0.934073,-0.0503387],[1,-1,-3,0],[9E+09,9E+09,9E+09,9E+09,9E+09,9E+09]], v5, seam13, weld13\Weave:=weave1, z1, tWeldGun;
		ArcLEnd [[-424.81,948.99,-7.39],[0.166172,-0.662098,-0.696056,-0.222531],[1,0,-2,0],[9E+09,9E+09,9E+09,9E+09,9E+09,9E+09]], v5, seam13, weld13\Weave:=weave1, fine, tWeldGun;
		MoveL [[-432.50,895.49,94.61],[0.171308,-0.660838,-0.695601,-0.2238],[1,0,-2,0],[9E+09,9E+09,9E+09,9E+09,9E+09,9E+09]], vmax, z0, tWeldGun;
		MoveL [[-428.23,950.42,262.61],[0.171376,-0.660832,-0.695567,-0.223872],[1,0,2,0],[9E+09,9E+09,9E+09,9E+09,9E+09,9E+09]], vmax, z0, tWeldGun;
		MoveJ [[-1240.64,940.49,246.51],[0.200371,-0.594607,-0.764476,-0.147887],[1,0,2,0],[9E+09,9E+09,9E+09,9E+09,9E+09,9E+09]], vmax, z0, tWeldGun;
		MoveL [[-1259.54,939.02,-1.77],[0.21012,-0.673416,-0.681865,-0.193445],[1,0,2,0],[9E+09,9E+09,9E+09,9E+09,9E+09,9E+09]], v100, z0, tWeldGun;
		ArcLStart [[-1260.55,943.84,-5.19],[0.210119,-0.673431,-0.681846,-0.19346],[1,0,2,0],[9E+09,9E+09,9E+09,9E+09,9E+09,9E+09]], v30, seam13, weld13\Weave:=weave1, fine, tWeldGun;
		ArcL [[-1288.10,948.60,-5.01],[0.116092,0.902251,0.0966143,0.403897],[1,0,3,0],[9E+09,9E+09,9E+09,9E+09,9E+09,9E+09]], v5, seam13, weld13\Weave:=weave1, z1, tWeldGun;
		ArcLEnd [[-1288.96,971.69,-6.42],[0.116097,0.902249,0.0965949,0.403904],[1,0,3,0],[9E+09,9E+09,9E+09,9E+09,9E+09,9E+09]], v5, seam13, weld13\Weave:=weave1, fine, tWeldGun;
		MoveL [[-1282.96,979.96,80.63],[0.116018,0.902243,0.096661,0.403925],[1,0,3,0],[9E+09,9E+09,9E+09,9E+09,9E+09,9E+09]], vmax, z0, tWeldGun;
		MoveJ [[-1358.53,1155.99,133.80],[0.133739,0.955506,0.10811,0.239657],[1,0,3,0],[9E+09,9E+09,9E+09,9E+09,9E+09,9E+09]], vmax, z0, tWeldGun;
		MoveL [[-1362.74,1158.80,0.21],[0.0670489,0.939872,-0.00304011,0.334868],[1,0,3,0],[9E+09,9E+09,9E+09,9E+09,9E+09,9E+09]], vmax, z0, tWeldGun;
		ArcLStart [[-1353.40,1155.11,-7.49],[0.0671234,0.939875,-0.00307785,0.334846],[1,0,3,0],[9E+09,9E+09,9E+09,9E+09,9E+09,9E+09]], v30, seam13, weld13\Weave:=weave1, fine, tWeldGun;
		ArcL [[-1354.09,1176.19,-7.46],[0.067105,0.939847,-0.0029865,0.334926],[1,0,3,0],[9E+09,9E+09,9E+09,9E+09,9E+09,9E+09]], v5, seam13, weld13\Weave:=weave1, z1, tWeldGun;
		ArcLEnd [[-1334.59,1191.37,-6.43],[0.222218,0.801402,-0.520283,0.194113],[1,0,4,0],[9E+09,9E+09,9E+09,9E+09,9E+09,9E+09]], v5, seam13, weld13\Weave:=weave1, fine, tWeldGun;
		MoveL [[-1328.99,1198.21,13.92],[0.263465,0.723639,-0.589044,0.244868],[1,0,4,0],[9E+09,9E+09,9E+09,9E+09,9E+09,9E+09]], v100, z0, tWeldGun;
		MoveL [[-1329.56,1242.98,151.23],[0.276586,0.758563,-0.567487,0.161373],[1,0,4,0],[9E+09,9E+09,9E+09,9E+09,9E+09,9E+09]], vmax, z0, tWeldGun;
		MoveJ [[-495.18,1248.58,261.21],[0.287177,0.742929,-0.58422,0.155801],[1,0,-1,0],[9E+09,9E+09,9E+09,9E+09,9E+09,9E+09]], vmax, z0, tWeldGun;
		MoveL [[-498.43,1204.30,4.59],[0.287207,0.742912,-0.584227,0.155798],[1,0,-1,0],[9E+09,9E+09,9E+09,9E+09,9E+09,9E+09]], vmax, z0, tWeldGun;
		ArcLStart [[-498.75,1196.41,-6.79],[0.287224,0.742903,-0.58423,0.155802],[1,0,-1,0],[9E+09,9E+09,9E+09,9E+09,9E+09,9E+09]], v30, seam13, weld13\Weave:=weave1, fine, tWeldGun;
		ArcL [[-476.78,1198.77,-9.23],[0.212945,0.671252,-0.679702,0.205135],[1,-1,0,0],[9E+09,9E+09,9E+09,9E+09,9E+09,9E+09]], v5, seam13, weld13\Weave:=weave1, z1, tWeldGun;
		SingArea\Wrist;
		ArcLEnd [[-463.84,1168.95,-10.12],[0.359543,0.0380909,-0.931217,-0.0459829],[1,-1,1,0],[9E+09,9E+09,9E+09,9E+09,9E+09,9E+09]], v5, seam13, weld13\Weave:=weave1, fine, tWeldGun;
		MoveL [[-421.44,1139.09,130.73],[0.359544,0.0381675,-0.931204,-0.0461746],[1,-1,1,0],[9E+09,9E+09,9E+09,9E+09,9E+09,9E+09]], vmax, z0, tWeldGun;
		MoveJ [[-409.78,718.78,85.27],[0.233728,0.658735,-0.674888,0.236571],[1,-1,0,0],[9E+09,9E+09,9E+09,9E+09,9E+09,9E+09]], vmax, z0, tWeldGun;
		MoveL [[-412.64,721.99,2.40],[0.233733,0.658767,-0.674882,0.236495],[1,-1,0,0],[9E+09,9E+09,9E+09,9E+09,9E+09,9E+09]], vmax, z0, tWeldGun;
		ArcLStart [[-411.66,717.54,-5.65],[0.233665,0.658899,-0.674713,0.236676],[1,-1,0,0],[9E+09,9E+09,9E+09,9E+09,9E+09,9E+09]], v30, seam13, weld13\Weave:=weave1, fine, tWeldGun;
		ArcLEnd [[-431.86,717.55,-6.04],[0.233667,0.658893,-0.674715,0.236685],[1,-1,0,0],[9E+09,9E+09,9E+09,9E+09,9E+09,9E+09]], v5, seam13, weld13\Weave:=weave1, fine, tWeldGun;
		MoveL [[-431.23,713.88,96.49],[0.233747,0.658736,-0.674884,0.236564],[1,-1,0,0],[9E+09,9E+09,9E+09,9E+09,9E+09,9E+09]], vmax, z0, tWeldGun;
		MoveL [[-1257.57,713.89,96.49],[0.233748,0.658741,-0.67488,0.236557],[1,-1,0,0],[9E+09,9E+09,9E+09,9E+09,9E+09,9E+09]], vmax, z0, tWeldGun;
		MoveL [[-1261.90,718.36,0.85],[0.233781,0.658746,-0.674869,0.236543],[1,-1,0,0],[9E+09,9E+09,9E+09,9E+09,9E+09,9E+09]], vmax, z0, tWeldGun;
		ArcLStart [[-1262.02,714.40,-4.57],[0.233749,0.658748,-0.674859,0.236598],[1,-1,0,0],[9E+09,9E+09,9E+09,9E+09,9E+09,9E+09]], v30, seam13, weld13\Weave:=weave1, fine, tWeldGun;
		ArcLEnd [[-1283.63,714.45,-4.57],[0.233759,0.658754,-0.674859,0.236572],[1,-1,0,0],[9E+09,9E+09,9E+09,9E+09,9E+09,9E+09]], v5, seam13, weld13\Weave:=weave1, fine, tWeldGun;
		MoveL [[-1282.90,713.31,123.57],[0.233803,0.658736,-0.674861,0.236572],[1,-1,0,0],[9E+09,9E+09,9E+09,9E+09,9E+09,9E+09]], vmax, z0, tWeldGun;
		MoveJ [[-1344.23,1422.02,101.83],[0.226991,-0.675391,-0.661326,-0.234461],[1,0,-2,0],[9E+09,9E+09,9E+09,9E+09,9E+09,9E+09]], vmax, z0, tWeldGun;
		MoveL [[-1344.24,1422.02,-3.62],[0.226998,-0.675396,-0.66132,-0.234453],[1,0,-2,0],[9E+09,9E+09,9E+09,9E+09,9E+09,9E+09]], vmax, z0, tWeldGun;
		ArcLStart [[-1344.81,1426.24,-8.72],[0.226999,-0.675402,-0.661313,-0.234454],[1,0,-2,0],[9E+09,9E+09,9E+09,9E+09,9E+09,9E+09]], v30, seam13, weld13\Weave:=weave1, fine, tWeldGun;
		ArcLEnd [[-1321.69,1425.45,-8.26],[0.227044,-0.675403,-0.661307,-0.234426],[1,0,-2,0],[9E+09,9E+09,9E+09,9E+09,9E+09,9E+09]], v5, seam13, weld13\Weave:=weave1, fine, tWeldGun;
		MoveL [[-1320.89,1427.11,81.12],[0.226982,-0.675417,-0.661301,-0.234462],[1,0,-2,0],[9E+09,9E+09,9E+09,9E+09,9E+09,9E+09]], vmax, z0, tWeldGun;
		MoveL [[-494.97,1419.41,70.78],[0.226989,-0.675424,-0.661294,-0.234454],[1,0,-2,0],[9E+09,9E+09,9E+09,9E+09,9E+09,9E+09]], vmax, z0, tWeldGun;
		MoveL [[-494.98,1419.41,-5.90],[0.226987,-0.675436,-0.661284,-0.23445],[1,0,-2,0],[9E+09,9E+09,9E+09,9E+09,9E+09,9E+09]], vmax, z0, tWeldGun;
		ArcLStart [[-493.66,1426.09,-11.11],[0.226969,-0.675494,-0.661234,-0.234443],[1,0,-2,0],[9E+09,9E+09,9E+09,9E+09,9E+09,9E+09]], v30, seam13, weld13\Weave:=weave1, fine, tWeldGun;
		ArcLEnd [[-472.90,1426.55,-9.92],[0.226962,-0.675517,-0.661214,-0.23444],[1,0,-2,0],[9E+09,9E+09,9E+09,9E+09,9E+09,9E+09]], v5, seam13, weld13\Weave:=weave1, fine, tWeldGun;
		MoveL [[-196.11,1086.38,621.33],[0.226996,-0.675454,-0.661218,-0.234578],[1,0,-2,0],[9E+09,9E+09,9E+09,9E+09,9E+09,9E+09]], vmax, z0, tWeldGun;

		!code ends here

        MoveJ pSafeS1, vmax, z10, tWeldGun;
	ENDPROC


